LIN {X 0,Y 130.565,Z 392.696,A -85,B 0,C 180,E1 -26244.314,E2 -26244.314} C_VEL
LIN {X 0,Y 127.932,Z 388.905,A -85,B 0,C 180,E1 -26247.47,E2 -26247.47} C_VEL
LIN {X 0,Y 124.893,Z 385.428,A -85,B 0,C 180,E1 -26251.722,E2 -26251.722} C_VEL
LIN {X 0,Y 123.933,Z 383.506,A -85,B 0,C 180,E1 -26253.474,E2 -26253.474} C_VEL
LIN {X 0,Y 121.317,Z 381.44,A -85,B 0,C 180,E1 -26258.762,E2 -26258.762} C_VEL
LIN {X 0,Y 119.958,Z 378.25,A -85,B 0,C 180,E1 -26264.062,E2 -26264.062} C_VEL
LIN {X 0,Y 119.864,Z 377.879,A -85,B 0,C 180,E1 -26264.703,E2 -26264.703} C_VEL
LIN {X 0,Y 119.859,Z 377.69,A -85,B 0,C 180,E1 -26276.64,E2 -26276.64} C_VEL
LIN {X 0,Y 120.448,Z 377.843,A -85,B 0,C 180,E1 -26279.061,E2 -26279.061} C_VEL
LIN {X 0,Y 121.379,Z 380.802,A -85,B 0,C 180,E1 -26282.646,E2 -26282.646} C_VEL
LIN {X 0,Y 123.476,Z 382.974,A -85,B 0,C 180,E1 -26287.153,E2 -26287.153} C_VEL
LIN {X 0,Y 124.269,Z 383.517,A -85,B 0,C 180,E1 -26288.487,E2 -26288.487} C_VEL
LIN {X 0,Y 126.216,Z 386.94,A -85,B 0,C 180,E1 -26291.712,E2 -26291.712} C_VEL
LIN {X 0,Y 128.213,Z 389.093,A -85,B 0,C 180,E1 -26294.339,E2 -26294.339} C_VEL
LIN {X 0,Y 131.436,Z 393.757,A -85,B 0,C 180,E1 -26298.071,E2 -26298.071} C_VEL
LIN {X 0,Y 134.937,Z 398.949,A -85,B 0,C 180,E1 -26301.484,E2 -26301.484} C_VEL
LIN {X 0,Y 138.77,Z 404.783,A -85,B 0,C 180,E1 -26304.698,E2 -26304.698} C_VEL
LIN {X 0,Y 143.672,Z 413.223,A -85,B 0,C 180,E1 -26308.311,E2 -26308.311} C_VEL
LIN {X 0,Y 147.61,Z 423.228,A -85,B 0,C 180,E1 -26311.147,E2 -26311.147} C_VEL
LIN {X 0,Y 151.744,Z 435.74,A -85,B 0,C 180,E1 -26313.948,E2 -26313.948} C_VEL
LIN {X 0,Y 152.367,Z 437.977,A -85,B 0,C 180,E1 -26314.368,E2 -26314.368} C_VEL
LIN {X 0,Y 147.684,Z 494.344,A -85,B 0,C 180,E1 -26316.574,E2 -26316.574} C_VEL
LIN {X 0,Y 145.389,Z 508.708,A -85,B 0,C 180,E1 -26317.524,E2 -26317.524} C_VEL
LIN {X 0,Y 142.287,Z 522.638,A -85,B 0,C 180,E1 -26318.924,E2 -26318.924} C_VEL
LIN {X 0,Y 138.683,Z 534.674,A -85,B 0,C 180,E1 -26320.519,E2 -26320.519} C_VEL
LIN {X 0,Y 134.203,Z 547.477,A -85,B 0,C 180,E1 -26322.845,E2 -26322.845} C_VEL
LIN {X 0,Y 130.787,Z 556.168,A -85,B 0,C 180,E1 -26324.873,E2 -26324.873} C_VEL
LIN {X 0,Y 126.494,Z 565.822,A -85,B 0,C 180,E1 -26327.646,E2 -26327.646} C_VEL
LIN {X 0,Y 121.378,Z 576.257,A -85,B 0,C 180,E1 -26331.502,E2 -26331.502} C_VEL
LIN {X 0,Y 116.597,Z 585.681,A -85,B 0,C 180,E1 -26336.11,E2 -26336.11} C_VEL
LIN {X 0,Y 112.251,Z 594.067,A -85,B 0,C 180,E1 -26341.476,E2 -26341.476} C_VEL
LIN {X 0,Y 109.035,Z 600.953,A -85,B 0,C 180,E1 -26347.245,E2 -26347.245} C_VEL
LIN {X 0,Y 106.871,Z 606.138,A -85,B 0,C 180,E1 -26352.783,E2 -26352.783} C_VEL
LIN {X 0,Y 105.467,Z 611.465,A -85,B 0,C 180,E1 -26360.407,E2 -26360.407} C_VEL
LIN {X 0,Y 105.191,Z 614.408,A -85,B 0,C 180,E1 -26366.166,E2 -26366.166} C_VEL
LIN {X 0,Y 105.389,Z 615.906,A -85,B 0,C 180,E1 -26369.997,E2 -26369.997} C_VEL
LIN {X 0,Y 105.237,Z 617.007,A -85,B 0,C 180,E1 -26373.826,E2 -26373.826} C_VEL
LIN {X 0,Y 105.699,Z 618.187,A -85,B 0,C 180,E1 -26381.502,E2 -26381.502} C_VEL
LIN {X 0,Y 107.664,Z 618.07,A -85,B 0,C 180,E1 -26389.046,E2 -26389.046} C_VEL
LIN {X 0,Y 111.464,Z 616.681,A -85,B 0,C 180,E1 -26396.187,E2 -26396.187} C_VEL
LIN {X 0,Y 116.761,Z 613.987,A -85,B 0,C 180,E1 -26402.797,E2 -26402.797} C_VEL
LIN {X 0,Y 123.623,Z 609.914,A -85,B 0,C 180,E1 -26408.704,E2 -26408.704} C_VEL
LIN {X 0,Y 131.691,Z 604.349,A -85,B 0,C 180,E1 -26413.925,E2 -26413.925} C_VEL
LIN {X 0,Y 135.186,Z 601.698,A -85,B 0,C 180,E1 -26415.806,E2 -26415.806} C_VEL
LIN {X 0,Y 138.09,Z 599.07,A -85,B 0,C 180,E1 -26417.662,E2 -26417.662} C_VEL
LIN {X 0,Y 141.798,Z 594.527,A -85,B 0,C 180,E1 -26420.954,E2 -26420.954} C_VEL
LIN {X 0,Y 145.772,Z 589.525,A -85,B 0,C 180,E1 -26423.968,E2 -26423.968} C_VEL
LIN {X 0,Y 148.969,Z 586.107,A -85,B 0,C 180,E1 -26425.363,E2 -26425.363} C_VEL
LIN {X 0,Y 157.532,Z 576.958,A -85,B 0,C 180,E1 -26427.952,E2 -26427.952} C_VEL
LIN {X 0,Y 166.118,Z 566.304,A -85,B 0,C 180,E1 -26430.141,E2 -26430.141} C_VEL
LIN {X 0,Y 174.249,Z 554.394,A -85,B 0,C 180,E1 -26431.914,E2 -26431.914} C_VEL
LIN {X 0,Y 181.076,Z 542.412,A -85,B 0,C 180,E1 -26433.207,E2 -26433.207} C_VEL
LIN {X 0,Y 187.168,Z 529.101,A -85,B 0,C 180,E1 -26434.308,E2 -26434.308} C_VEL
LIN {X 0,Y 192.216,Z 515.011,A -85,B 0,C 180,E1 -26435.118,E2 -26435.118} C_VEL
LIN {X 0,Y 196.051,Z 500.312,A -85,B 0,C 180,E1 -26435.708,E2 -26435.708} C_VEL
LIN {X 0,Y 198.473,Z 485.503,A -85,B 0,C 180,E1 -26436.14,E2 -26436.14} C_VEL
LIN {X 0,Y 199.396,Z 476.925,A -85,B 0,C 180,E1 -26436.363,E2 -26436.363} C_VEL
LIN {X 0,Y 198.019,Z 472.232,A -85,B 0,C 180,E1 -26438.547,E2 -26438.547} C_VEL
LIN {X 0,Y 196.974,Z 468.88,A -85,B 0,C 180,E1 -26440.498,E2 -26440.498} C_VEL
LIN {X 0,Y 195.91,Z 465.386,A -85,B 0,C 180,E1 -26443.053,E2 -26443.053} C_VEL
LIN {X 0,Y 195.243,Z 463.284,A -85,B 0,C 180,E1 -26445.138,E2 -26445.138} C_VEL
LIN {X 0,Y 194.3,Z 461.074,A -85,B 0,C 180,E1 -26451.68,E2 -26451.68} C_VEL
LIN {X 0,Y 195.325,Z 463.03,A -85,B 0,C 180,E1 -26457.55,E2 -26457.55} C_VEL
LIN {X 0,Y 196.809,Z 466.839,A -85,B 0,C 180,E1 -26461.401,E2 -26461.401} C_VEL
LIN {X 0,Y 198.529,Z 470.876,A -85,B 0,C 180,E1 -26464.413,E2 -26464.413} C_VEL
LIN {X 0,Y 199.707,Z 473.742,A -85,B 0,C 180,E1 -26466.094,E2 -26466.094} C_VEL
LIN {X 0,Y 197.371,Z 491.479,A -85,B 0,C 180,E1 -26466.567,E2 -26466.567} C_VEL
LIN {X 0,Y 194.393,Z 504.956,A -85,B 0,C 180,E1 -26467.115,E2 -26467.115} C_VEL
LIN {X 0,Y 189.943,Z 519.303,A -85,B 0,C 180,E1 -26467.963,E2 -26467.963} C_VEL
LIN {X 0,Y 184.163,Z 533.238,A -85,B 0,C 180,E1 -26469.107,E2 -26469.107} C_VEL
LIN {X 0,Y 177.795,Z 545.567,A -85,B 0,C 180,E1 -26470.508,E2 -26470.508} C_VEL
LIN {X 0,Y 170.279,Z 557.457,A -85,B 0,C 180,E1 -26472.235,E2 -26472.235} C_VEL
LIN {X 0,Y 163.039,Z 567.153,A -85,B 0,C 180,E1 -26474.107,E2 -26474.107} C_VEL
LIN {X 0,Y 155.175,Z 576.173,A -85,B 0,C 180,E1 -26476.356,E2 -26476.356} C_VEL
LIN {X 0,Y 146.298,Z 584.96,A -85,B 0,C 180,E1 -26479.346,E2 -26479.346} C_VEL
LIN {X 0,Y 137.329,Z 592.535,A -85,B 0,C 180,E1 -26482.91,E2 -26482.91} C_VEL
LIN {X 0,Y 129.687,Z 598.111,A -85,B 0,C 180,E1 -26486.606,E2 -26486.606} C_VEL
LIN {X 0,Y 121.78,Z 603.078,A -85,B 0,C 180,E1 -26491.29,E2 -26491.29} C_VEL
LIN {X 0,Y 114.351,Z 606.986,A -85,B 0,C 180,E1 -26496.973,E2 -26496.973} C_VEL
LIN {X 0,Y 107.549,Z 609.772,A -85,B 0,C 180,E1 -26504.048,E2 -26504.048} C_VEL
LIN {X 0,Y 102.478,Z 611.008,A -85,B 0,C 180,E1 -26511.891,E2 -26511.891} C_VEL
LIN {X 0,Y 99.227,Z 610.742,A -85,B 0,C 180,E1 -26520.282,E2 -26520.282} C_VEL
LIN {X 0,Y 97.751,Z 608.962,A -85,B 0,C 180,E1 -26529.17,E2 -26529.17} C_VEL
LIN {X 0,Y 97.864,Z 605.87,A -85,B 0,C 180,E1 -26537.562,E2 -26537.562} C_VEL
LIN {X 0,Y 98.97,Z 602.563,A -85,B 0,C 180,E1 -26543.788,E2 -26543.788} C_VEL
LIN {X 0,Y 100.796,Z 598.268,A -85,B 0,C 180,E1 -26550.004,E2 -26550.004} C_VEL
LIN {X 0,Y 103.829,Z 592.06,A -85,B 0,C 180,E1 -26556.806,E2 -26556.806} C_VEL
LIN {X 0,Y 107.94,Z 584.679,A -85,B 0,C 180,E1 -26562.874,E2 -26562.874} C_VEL
LIN {X 0,Y 112.553,Z 576.205,A -85,B 0,C 180,E1 -26568.196,E2 -26568.196} C_VEL
LIN {X 0,Y 117.725,Z 566.442,A -85,B 0,C 180,E1 -26572.836,E2 -26572.836} C_VEL
LIN {X 0,Y 123.092,Z 555.588,A -85,B 0,C 180,E1 -26576.723,E2 -26576.723} C_VEL
LIN {X 0,Y 128.33,Z 543.576,A -85,B 0,C 180,E1 -26579.985,E2 -26579.985} C_VEL
LIN {X 0,Y 133.128,Z 530.85,A -85,B 0,C 180,E1 -26582.567,E2 -26582.567} C_VEL
LIN {X 0,Y 137.139,Z 517.829,A -85,B 0,C 180,E1 -26584.539,E2 -26584.539} C_VEL
LIN {X 0,Y 140.486,Z 503.558,A -85,B 0,C 180,E1 -26586.115,E2 -26586.115} C_VEL
LIN {X 0,Y 142.816,Z 489.892,A -85,B 0,C 180,E1 -26587.138,E2 -26587.138} C_VEL
LIN {X 0,Y 144.553,Z 473.342,A -85,B 0,C 180,E1 -26587.883,E2 -26587.883} C_VEL
LIN {X 0,Y 147.842,Z 434.546,A -85,B 0,C 180,E1 -26589.335,E2 -26589.335} C_VEL
LIN {X 0,Y 143.5,Z 424.674,A -85,B 0,C 180,E1 -26592.28,E2 -26592.28} C_VEL
LIN {X 0,Y 138.696,Z 415.374,A -85,B 0,C 180,E1 -26595.804,E2 -26595.804} C_VEL
LIN {X 0,Y 133.828,Z 407.051,A -85,B 0,C 180,E1 -26599.922,E2 -26599.922} C_VEL
LIN {X 0,Y 130.389,Z 401.996,A -85,B 0,C 180,E1 -26603.29,E2 -26603.29} C_VEL
LIN {X 0,Y 128.308,Z 398.785,A -85,B 0,C 180,E1 -26605.658,E2 -26605.658} C_VEL
LIN {X 0,Y 125.687,Z 394.914,A -85,B 0,C 180,E1 -26609.089,E2 -26609.089} C_VEL
LIN {X 0,Y 123.305,Z 392.01,A -85,B 0,C 180,E1 -26612.724,E2 -26612.724} C_VEL
LIN {X 0,Y 122.54,Z 390.343,A -85,B 0,C 180,E1 -26614.234,E2 -26614.234} C_VEL
LIN {X 0,Y 120.138,Z 388.287,A -85,B 0,C 180,E1 -26619.453,E2 -26619.453} C_VEL
LIN {X 0,Y 118.826,Z 384.875,A -85,B 0,C 180,E1 -26625.443,E2 -26625.443} C_VEL
LIN {X 0,Y 119.141,Z 384.732,A -85,B 0,C 180,E1 -26637.465,E2 -26637.465} C_VEL
LIN {X 0,Y 119.373,Z 385.115,A -85,B 0,C 180,E1 -26638.563,E2 -26638.563} C_VEL
LIN {X 0,Y 120.443,Z 388.08,A -85,B 0,C 180,E1 -26642.666,E2 -26642.666} C_VEL
LIN {X 0,Y 122.798,Z 390.406,A -85,B 0,C 180,E1 -26647.639,E2 -26647.639} C_VEL
LIN {X 0,Y 124.835,Z 393.821,A -85,B 0,C 180,E1 -26651.142,E2 -26651.142} C_VEL
LIN {X 0,Y 126.414,Z 395.654,A -85,B 0,C 180,E1 -26653.346,E2 -26653.346} C_VEL
LIN {X 0,Y 129.348,Z 400.172,A -85,B 0,C 180,E1 -26657.001,E2 -26657.001} C_VEL
LIN {X 0,Y 132.297,Z 404.722,A -85,B 0,C 180,E1 -26660.1,E2 -26660.1} C_VEL
LIN {X 0,Y 135.761,Z 410.198,A -85,B 0,C 180,E1 -26663.251,E2 -26663.251} C_VEL
LIN {X 0,Y 140.215,Z 418.181,A -85,B 0,C 180,E1 -26666.816,E2 -26666.816} C_VEL
LIN {X 0,Y 143.851,Z 427.962,A -85,B 0,C 180,E1 -26669.649,E2 -26669.649} C_VEL
LIN {X 0,Y 147.514,Z 439.791,A -85,B 0,C 180,E1 -26672.38,E2 -26672.38} C_VEL
LIN {X 0,Y 142.873,Z 493.821,A -85,B 0,C 180,E1 -26674.515,E2 -26674.515} C_VEL
LIN {X 0,Y 140.487,Z 508.265,A -85,B 0,C 180,E1 -26675.46,E2 -26675.46} C_VEL
LIN {X 0,Y 137.276,Z 522.25,A -85,B 0,C 180,E1 -26676.872,E2 -26676.872} C_VEL
LIN {X 0,Y 132.944,Z 536.105,A -85,B 0,C 180,E1 -26678.759,E2 -26678.759} C_VEL
LIN {X 0,Y 128.467,Z 548.145,A -85,B 0,C 180,E1 -26681.033,E2 -26681.033} C_VEL
LIN {X 0,Y 123.348,Z 559.998,A -85,B 0,C 180,E1 -26683.996,E2 -26683.996} C_VEL
LIN {X 0,Y 117.775,Z 571.436,A -85,B 0,C 180,E1 -26687.827,E2 -26687.827} C_VEL
LIN {X 0,Y 112.305,Z 581.637,A -85,B 0,C 180,E1 -26692.396,E2 -26692.396} C_VEL
LIN {X 0,Y 107.744,Z 590.107,A -85,B 0,C 180,E1 -26697.439,E2 -26697.439} C_VEL
LIN {X 0,Y 103.985,Z 597.14,A -85,B 0,C 180,E1 -26702.854,E2 -26702.854} C_VEL
LIN {X 0,Y 100.736,Z 603.799,A -85,B 0,C 180,E1 -26709.58,E2 -26709.58} C_VEL
LIN {X 0,Y 98.674,Z 609.674,A -85,B 0,C 180,E1 -26717.659,E2 -26717.659} C_VEL
LIN {X 0,Y 98.264,Z 611.989,A -85,B 0,C 180,E1 -26721.772,E2 -26721.772} C_VEL
LIN {X 0,Y 98.308,Z 615.447,A -85,B 0,C 180,E1 -26729.996,E2 -26729.996} C_VEL
LIN {X 0,Y 98.155,Z 616.589,A -85,B 0,C 180,E1 -26734.102,E2 -26734.102} C_VEL
LIN {X 0,Y 98.71,Z 617.854,A -85,B 0,C 180,E1 -26742.329,E2 -26742.329} C_VEL
LIN {X 0,Y 100.934,Z 617.823,A -85,B 0,C 180,E1 -26750.37,E2 -26750.37} C_VEL
LIN {X 0,Y 105.094,Z 616.524,A -85,B 0,C 180,E1 -26757.908,E2 -26757.908} C_VEL
LIN {X 0,Y 110.842,Z 613.932,A -85,B 0,C 180,E1 -26764.791,E2 -26764.791} C_VEL
LIN {X 0,Y 118.143,Z 609.985,A -85,B 0,C 180,E1 -26770.867,E2 -26770.867} C_VEL
LIN {X 0,Y 126.657,Z 604.538,A -85,B 0,C 180,E1 -26776.161,E2 -26776.161} C_VEL
LIN {X 0,Y 133.774,Z 599.397,A -85,B 0,C 180,E1 -26779.616,E2 -26779.616} C_VEL
LIN {X 0,Y 142.665,Z 592.072,A -85,B 0,C 180,E1 -26783.174,E2 -26783.174} C_VEL
LIN {X 0,Y 148.969,Z 586.107,A -85,B 0,C 180,E1 -26785.363,E2 -26785.363} C_VEL
LIN {X 0,Y 152.163,Z 582.553,A -85,B 0,C 180,E1 -26786.685,E2 -26786.685} C_VEL
LIN {X 0,Y 156.304,Z 576.602,A -85,B 0,C 180,E1 -26789.221,E2 -26789.221} C_VEL
LIN {X 0,Y 160.479,Z 570.287,A -85,B 0,C 180,E1 -26791.519,E2 -26791.519} C_VEL
LIN {X 0,Y 163.59,Z 566.039,A -85,B 0,C 180,E1 -26792.464,E2 -26792.464} C_VEL
LIN {X 0,Y 171.828,Z 554.28,A -85,B 0,C 180,E1 -26794.13,E2 -26794.13} C_VEL
LIN {X 0,Y 178.803,Z 542.339,A -85,B 0,C 180,E1 -26795.354,E2 -26795.354} C_VEL
LIN {X 0,Y 185.017,Z 529.103,A -85,B 0,C 180,E1 -26796.4,E2 -26796.4} C_VEL
LIN {X 0,Y 190.172,Z 515.088,A -85,B 0,C 180,E1 -26797.154,E2 -26797.154} C_VEL
LIN {X 0,Y 193.988,Z 500.922,A -85,B 0,C 180,E1 -26797.696,E2 -26797.696} C_VEL
LIN {X 0,Y 196.522,Z 486.259,A -85,B 0,C 180,E1 -26798.109,E2 -26798.109} C_VEL
LIN {X 0,Y 197.129,Z 480.708,A -85,B 0,C 180,E1 -26798.293,E2 -26798.293} C_VEL
LIN {X 0,Y 195.702,Z 475.495,A -85,B 0,C 180,E1 -26801.142,E2 -26801.142} C_VEL
LIN {X 0,Y 194.724,Z 471.967,A -85,B 0,C 180,E1 -26803.756,E2 -26803.756} C_VEL
LIN {X 0,Y 194.117,Z 470.099,A -85,B 0,C 180,E1 -26805.854,E2 -26805.854} C_VEL
LIN {X 0,Y 193.405,Z 468.125,A -85,B 0,C 180,E1 -26811.642,E2 -26811.642} C_VEL
LIN {X 0,Y 194.291,Z 469.945,A -85,B 0,C 180,E1 -26817.148,E2 -26817.148} C_VEL
LIN {X 0,Y 195.675,Z 473.82,A -85,B 0,C 180,E1 -26821.02,E2 -26821.02} C_VEL
LIN {X 0,Y 197.375,Z 478.057,A -85,B 0,C 180,E1 -26824.16,E2 -26824.16} C_VEL
LIN {X 0,Y 195.492,Z 491.681,A -85,B 0,C 180,E1 -26824.575,E2 -26824.575} C_VEL
LIN {X 0,Y 192.282,Z 505.823,A -85,B 0,C 180,E1 -26825.124,E2 -26825.124} C_VEL
LIN {X 0,Y 187.68,Z 520.146,A -85,B 0,C 180,E1 -26825.946,E2 -26825.946} C_VEL
LIN {X 0,Y 182.297,Z 532.862,A -85,B 0,C 180,E1 -26826.935,E2 -26826.935} C_VEL
LIN {X 0,Y 175.759,Z 545.305,A -85,B 0,C 180,E1 -26828.262,E2 -26828.262} C_VEL
LIN {X 0,Y 168.052,Z 557.274,A -85,B 0,C 180,E1 -26829.909,E2 -26829.909} C_VEL
LIN {X 0,Y 159.79,Z 567.991,A -85,B 0,C 180,E1 -26831.884,E2 -26831.884} C_VEL
LIN {X 0,Y 152.067,Z 576.524,A -85,B 0,C 180,E1 -26833.953,E2 -26833.953} C_VEL
LIN {X 0,Y 143.374,Z 584.837,A -85,B 0,C 180,E1 -26836.675,E2 -26836.675} C_VEL
LIN {X 0,Y 134.546,Z 592.07,A -85,B 0,C 180,E1 -26839.92,E2 -26839.92} C_VEL
LIN {X 0,Y 126.152,Z 597.976,A -85,B 0,C 180,E1 -26843.63,E2 -26843.63} C_VEL
LIN {X 0,Y 116.987,Z 603.443,A -85,B 0,C 180,E1 -26848.723,E2 -26848.723} C_VEL
LIN {X 0,Y 109.905,Z 606.939,A -85,B 0,C 180,E1 -26853.774,E2 -26853.774} C_VEL
LIN {X 0,Y 102.361,Z 609.85,A -85,B 0,C 180,E1 -26860.959,E2 -26860.959} C_VEL
LIN {X 0,Y 96.569,Z 611.237,A -85,B 0,C 180,E1 -26869.086,E2 -26869.086} C_VEL
LIN {X 0,Y 92.708,Z 611.122,A -85,B 0,C 180,E1 -26877.955,E2 -26877.955} C_VEL
LIN {X 0,Y 90.794,Z 609.529,A -85,B 0,C 180,E1 -26887.235,E2 -26887.235} C_VEL
LIN {X 0,Y 90.662,Z 606.49,A -85,B 0,C 180,E1 -26896.557,E2 -26896.557} C_VEL
LIN {X 0,Y 91.859,Z 602.883,A -85,B 0,C 180,E1 -26904.033,E2 -26904.033} C_VEL
LIN {X 0,Y 94.334,Z 597.49,A -85,B 0,C 180,E1 -26912.139,E2 -26912.139} C_VEL
LIN {X 0,Y 97.853,Z 591.02,A -85,B 0,C 180,E1 -26919.303,E2 -26919.303} C_VEL
LIN {X 0,Y 102.587,Z 582.975,A -85,B 0,C 180,E1 -26925.908,E2 -26925.908} C_VEL
LIN {X 0,Y 107.51,Z 574.56,A -85,B 0,C 180,E1 -26931.075,E2 -26931.075} C_VEL
LIN {X 0,Y 113.086,Z 564.432,A -85,B 0,C 180,E1 -26935.791,E2 -26935.791} C_VEL
LIN {X 0,Y 118.876,Z 553.081,A -85,B 0,C 180,E1 -26939.682,E2 -26939.682} C_VEL
LIN {X 0,Y 123.921,Z 541.774,A -85,B 0,C 180,E1 -26942.604,E2 -26942.604} C_VEL
LIN {X 0,Y 128.938,Z 528.539,A -85,B 0,C 180,E1 -26945.156,E2 -26945.156} C_VEL
LIN {X 0,Y 133.138,Z 514.65,A -85,B 0,C 180,E1 -26947.143,E2 -26947.143} C_VEL
LIN {X 0,Y 136.364,Z 500.569,A -85,B 0,C 180,E1 -26948.583,E2 -26948.583} C_VEL
LIN {X 0,Y 138.668,Z 486.383,A -85,B 0,C 180,E1 -26949.526,E2 -26949.526} C_VEL
LIN {X 0,Y 143.173,Z 436.992,A -85,B 0,C 180,E1 -26951.425,E2 -26951.425} C_VEL
LIN {X 0,Y 138.636,Z 426.756,A -85,B 0,C 180,E1 -26954.79,E2 -26954.79} C_VEL
LIN {X 0,Y 134.385,Z 418.447,A -85,B 0,C 180,E1 -26958.313,E2 -26958.313} C_VEL
LIN {X 0,Y 130.256,Z 411.423,A -85,B 0,C 180,E1 -26962.248,E2 -26962.248} C_VEL
LIN {X 0,Y 126.452,Z 405.272,A -85,B 0,C 180,E1 -26966.64,E2 -26966.64} C_VEL
LIN {X 0,Y 123.842,Z 401.369,A -85,B 0,C 180,E1 -26970.293,E2 -26970.293} C_VEL
LIN {X 0,Y 121.463,Z 398.016,A -85,B 0,C 180,E1 -26974.334,E2 -26974.334} C_VEL
LIN {X 0,Y 121.025,Z 397.131,A -85,B 0,C 180,E1 -26975.272,E2 -26975.272} C_VEL
LIN {X 0,Y 118.602,Z 394.472,A -85,B 0,C 180,E1 -26981.47,E2 -26981.47} C_VEL
LIN {X 0,Y 117.811,Z 391.858,A -85,B 0,C 180,E1 -26986.196,E2 -26986.196} C_VEL
LIN {X 0,Y 118.259,Z 391.878,A -85,B 0,C 180,E1 -26997.603,E2 -26997.603} C_VEL
LIN {X 0,Y 119.232,Z 394.875,A -85,B 0,C 180,E1 -27001.872,E2 -27001.872} C_VEL
LIN {X 0,Y 121.348,Z 397.207,A -85,B 0,C 180,E1 -27006.751,E2 -27006.751} C_VEL
LIN {X 0,Y 123.458,Z 400.701,A -85,B 0,C 180,E1 -27010.55,E2 -27010.55} C_VEL
LIN {X 0,Y 124.654,Z 402.238,A -85,B 0,C 180,E1 -27012.33,E2 -27012.33} C_VEL
LIN {X 0,Y 127.406,Z 406.711,A -85,B 0,C 180,E1 -27016.011,E2 -27016.011} C_VEL
LIN {X 0,Y 130.249,Z 411.318,A -85,B 0,C 180,E1 -27019.198,E2 -27019.198} C_VEL
LIN {X 0,Y 133.511,Z 416.904,A -85,B 0,C 180,E1 -27022.367,E2 -27022.367} C_VEL
LIN {X 0,Y 136.961,Z 423.54,A -85,B 0,C 180,E1 -27025.351,E2 -27025.351} C_VEL
LIN {X 0,Y 140.042,Z 432.268,A -85,B 0,C 180,E1 -27027.965,E2 -27027.965} C_VEL
LIN {X 0,Y 142.868,Z 441.747,A -85,B 0,C 180,E1 -27030.281,E2 -27030.281} C_VEL
LIN {X 0,Y 138.312,Z 492.874,A -85,B 0,C 180,E1 -27032.288,E2 -27032.288} C_VEL
LIN {X 0,Y 135.883,Z 507.41,A -85,B 0,C 180,E1 -27033.223,E2 -27033.223} C_VEL
LIN {X 0,Y 132.455,Z 521.863,A -85,B 0,C 180,E1 -27034.668,E2 -27034.668} C_VEL
LIN {X 0,Y 127.952,Z 535.743,A -85,B 0,C 180,E1 -27036.549,E2 -27036.549} C_VEL
LIN {X 0,Y 123.17,Z 548.031,A -85,B 0,C 180,E1 -27038.878,E2 -27038.878} C_VEL
LIN {X 0,Y 117.914,Z 559.668,A -85,B 0,C 180,E1 -27041.834,E2 -27041.834} C_VEL
LIN {X 0,Y 112.578,Z 570.177,A -85,B 0,C 180,E1 -27045.383,E2 -27045.383} C_VEL
LIN {X 0,Y 106.709,Z 580.573,A -85,B 0,C 180,E1 -27050.044,E2 -27050.044} C_VEL
LIN {X 0,Y 101.75,Z 589.176,A -85,B 0,C 180,E1 -27055.257,E2 -27055.257} C_VEL
LIN {X 0,Y 97.059,Z 597.36,A -85,B 0,C 180,E1 -27061.919,E2 -27061.919} C_VEL
LIN {X 0,Y 94.071,Z 603.1,A -85,B 0,C 180,E1 -27068.061,E2 -27068.061} C_VEL
LIN {X 0,Y 91.718,Z 609.076,A -85,B 0,C 180,E1 -27076.706,E2 -27076.706} C_VEL
LIN {X 0,Y 91.217,Z 611.437,A -85,B 0,C 180,E1 -27081.132,E2 -27081.132} C_VEL
LIN {X 0,Y 91.217,Z 614.987,A -85,B 0,C 180,E1 -27089.996,E2 -27089.996} C_VEL
LIN {X 0,Y 91.066,Z 616.171,A -85,B 0,C 180,E1 -27094.422,E2 -27094.422} C_VEL
LIN {X 0,Y 91.757,Z 617.52,A -85,B 0,C 180,E1 -27103.28,E2 -27103.28} C_VEL
LIN {X 0,Y 94.267,Z 617.573,A -85,B 0,C 180,E1 -27111.882,E2 -27111.882} C_VEL
LIN {X 0,Y 98.832,Z 616.364,A -85,B 0,C 180,E1 -27119.848,E2 -27119.848} C_VEL
LIN {X 0,Y 105.074,Z 613.869,A -85,B 0,C 180,E1 -27127.007,E2 -27127.007} C_VEL
LIN {X 0,Y 112.855,Z 610.028,A -85,B 0,C 180,E1 -27133.232,E2 -27133.232} C_VEL
LIN {X 0,Y 121.833,Z 604.723,A -85,B 0,C 180,E1 -27138.577,E2 -27138.577} C_VEL
LIN {X 0,Y 129.296,Z 599.641,A -85,B 0,C 180,E1 -27142.009,E2 -27142.009} C_VEL
LIN {X 0,Y 138.528,Z 592.437,A -85,B 0,C 180,E1 -27145.524,E2 -27145.524} C_VEL
LIN {X 0,Y 148.166,Z 583.599,A -85,B 0,C 180,E1 -27148.622,E2 -27148.622} C_VEL
LIN {X 0,Y 156.862,Z 574.366,A -85,B 0,C 180,E1 -27150.882,E2 -27150.882} C_VEL
LIN {X 0,Y 163.59,Z 566.039,A -85,B 0,C 180,E1 -27152.464,E2 -27152.464} C_VEL
LIN {X 0,Y 166.673,Z 561.678,A -85,B 0,C 180,E1 -27153.335,E2 -27153.335} C_VEL
LIN {X 0,Y 170.722,Z 554.474,A -85,B 0,C 180,E1 -27155.189,E2 -27155.189} C_VEL
LIN {X 0,Y 174.448,Z 546.9,A -85,B 0,C 180,E1 -27156.911,E2 -27156.911} C_VEL
LIN {X 0,Y 176.941,Z 541.962,A -85,B 0,C 180,E1 -27157.582,E2 -27157.582} C_VEL
LIN {X 0,Y 183.124,Z 529.102,A -85,B 0,C 180,E1 -27158.534,E2 -27158.534} C_VEL
LIN {X 0,Y 188.332,Z 515.305,A -85,B 0,C 180,E1 -27159.223,E2 -27159.223} C_VEL
LIN {X 0,Y 192.356,Z 500.713,A -85,B 0,C 180,E1 -27159.757,E2 -27159.757} C_VEL
LIN {X 0,Y 194.963,Z 485.994,A -85,B 0,C 180,E1 -27160.146,E2 -27160.146} C_VEL
LIN {X 0,Y 195.085,Z 484.899,A -85,B 0,C 180,E1 -27160.213,E2 -27160.213} C_VEL
LIN {X 0,Y 194.284,Z 481.515,A -85,B 0,C 180,E1 -27162.228,E2 -27162.228} C_VEL
LIN {X 0,Y 193.496,Z 478.254,A -85,B 0,C 180,E1 -27164.732,E2 -27164.732} C_VEL
LIN {X 0,Y 193.088,Z 477.008,A -85,B 0,C 180,E1 -27166.314,E2 -27166.314} C_VEL
LIN {X 0,Y 192.509,Z 475.192,A -85,B 0,C 180,E1 -27171.602,E2 -27171.602} C_VEL
LIN {X 0,Y 193.266,Z 476.862,A -85,B 0,C 180,E1 -27176.742,E2 -27176.742} C_VEL
LIN {X 0,Y 194.452,Z 480.465,A -85,B 0,C 180,E1 -27180.388,E2 -27180.388} C_VEL
LIN {X 0,Y 195.276,Z 482.796,A -85,B 0,C 180,E1 -27182.255,E2 -27182.255} C_VEL
LIN {X 0,Y 193.115,Z 495.782,A -85,B 0,C 180,E1 -27182.652,E2 -27182.652} C_VEL
LIN {X 0,Y 189.61,Z 509.454,A -85,B 0,C 180,E1 -27183.231,E2 -27183.231} C_VEL
LIN {X 0,Y 184.926,Z 522.764,A -85,B 0,C 180,E1 -27183.992,E2 -27183.992} C_VEL
LIN {X 0,Y 178.766,Z 536.319,A -85,B 0,C 180,E1 -27185.058,E2 -27185.058} C_VEL
LIN {X 0,Y 172.336,Z 547.773,A -85,B 0,C 180,E1 -27186.287,E2 -27186.287} C_VEL
LIN {X 0,Y 164.387,Z 559.452,A -85,B 0,C 180,E1 -27187.876,E2 -27187.876} C_VEL
LIN {X 0,Y 155.49,Z 570.334,A -85,B 0,C 180,E1 -27189.883,E2 -27189.883} C_VEL
LIN {X 0,Y 147.286,Z 578.835,A -85,B 0,C 180,E1 -27192.002,E2 -27192.002} C_VEL
LIN {X 0,Y 138.081,Z 587.013,A -85,B 0,C 180,E1 -27194.759,E2 -27194.759} C_VEL
LIN {X 0,Y 129.239,Z 593.716,A -85,B 0,C 180,E1 -27197.901,E2 -27197.901} C_VEL
LIN {X 0,Y 120.837,Z 599.162,A -85,B 0,C 180,E1 -27201.485,E2 -27201.485} C_VEL
LIN {X 0,Y 112.414,Z 603.82,A -85,B 0,C 180,E1 -27205.952,E2 -27205.952} C_VEL
LIN {X 0,Y 105.827,Z 606.892,A -85,B 0,C 180,E1 -27210.314,E2 -27210.314} C_VEL
LIN {X 0,Y 97.49,Z 609.929,A -85,B 0,C 180,E1 -27217.541,E2 -27217.541} C_VEL
LIN {X 0,Y 90.922,Z 611.436,A -85,B 0,C 180,E1 -27225.925,E2 -27225.925} C_VEL
LIN {X 0,Y 86.377,Z 611.466,A -85,B 0,C 180,E1 -27235.287,E2 -27235.287} C_VEL
LIN {X 0,Y 83.897,Z 610.021,A -85,B 0,C 180,E1 -27245.243,E2 -27245.243} C_VEL
LIN {X 0,Y 83.44,Z 608.743,A -85,B 0,C 180,E1 -27250.316,E2 -27250.316} C_VEL
LIN {X 0,Y 84.053,Z 605.08,A -85,B 0,C 180,E1 -27260.378,E2 -27260.378} C_VEL
LIN {X 0,Y 85.594,Z 601.369,A -85,B 0,C 180,E1 -27267.651,E2 -27267.651} C_VEL
LIN {X 0,Y 87.992,Z 596.701,A -85,B 0,C 180,E1 -27274.585,E2 -27274.585} C_VEL
LIN {X 0,Y 92.051,Z 589.969,A -85,B 0,C 180,E1 -27282.124,E2 -27282.124} C_VEL
LIN {X 0,Y 97.368,Z 581.584,A -85,B 0,C 180,E1 -27288.958,E2 -27288.958} C_VEL
LIN {X 0,Y 102.738,Z 572.829,A -85,B 0,C 180,E1 -27294.236,E2 -27294.236} C_VEL
LIN {X 0,Y 108.804,Z 562.214,A -85,B 0,C 180,E1 -27298.98,E2 -27298.98} C_VEL
LIN {X 0,Y 114.423,Z 551.482,A -85,B 0,C 180,E1 -27302.513,E2 -27302.513} C_VEL
LIN {X 0,Y 119.788,Z 539.763,A -85,B 0,C 180,E1 -27305.41,E2 -27305.41} C_VEL
LIN {X 0,Y 124.798,Z 526.675,A -85,B 0,C 180,E1 -27307.834,E2 -27307.834} C_VEL
LIN {X 0,Y 128.809,Z 513.594,A -85,B 0,C 180,E1 -27309.623,E2 -27309.623} C_VEL
LIN {X 0,Y 132.1,Z 499.36,A -85,B 0,C 180,E1 -27311.023,E2 -27311.023} C_VEL
LIN {X 0,Y 134.414,Z 484.873,A -85,B 0,C 180,E1 -27311.907,E2 -27311.907} C_VEL
LIN {X 0,Y 138.632,Z 439.572,A -85,B 0,C 180,E1 -27313.64,E2 -27313.64} C_VEL
LIN {X 0,Y 134.588,Z 430.258,A -85,B 0,C 180,E1 -27316.979,E2 -27316.979} C_VEL
LIN {X 0,Y 131.132,Z 423.275,A -85,B 0,C 180,E1 -27320.17,E2 -27320.17} C_VEL
LIN {X 0,Y 127.804,Z 417.282,A -85,B 0,C 180,E1 -27323.668,E2 -27323.668} C_VEL
LIN {X 0,Y 124.306,Z 411.372,A -85,B 0,C 180,E1 -27328.086,E2 -27328.086} C_VEL
LIN {X 0,Y 122.054,Z 407.807,A -85,B 0,C 180,E1 -27331.503,E2 -27331.503} C_VEL
LIN {X 0,Y 119.818,Z 404.229,A -85,B 0,C 180,E1 -27335.76,E2 -27335.76} C_VEL
LIN {X 0,Y 117.128,Z 400.289,A -85,B 0,C 180,E1 -27344.113,E2 -27344.113} C_VEL
LIN {X 0,Y 116.912,Z 399.034,A -85,B 0,C 180,E1 -27346.088,E2 -27346.088} C_VEL
LIN {X 0,Y 116.679,Z 398.767,A -85,B 0,C 180,E1 -27353.082,E2 -27353.082} C_VEL
LIN {X 0,Y 117.23,Z 398.988,A -85,B 0,C 180,E1 -27357.076,E2 -27357.076} C_VEL
LIN {X 0,Y 118.365,Z 402.176,A -85,B 0,C 180,E1 -27362.07,E2 -27362.07} C_VEL
LIN {X 0,Y 119.958,Z 404.022,A -85,B 0,C 180,E1 -27365.896,E2 -27365.896} C_VEL
LIN {X 0,Y 122.086,Z 407.575,A -85,B 0,C 180,E1 -27369.946,E2 -27369.946} C_VEL
LIN {X 0,Y 123.233,Z 409.368,A -85,B 0,C 180,E1 -27371.762,E2 -27371.762} C_VEL
LIN {X 0,Y 125.272,Z 412.815,A -85,B 0,C 180,E1 -27374.683,E2 -27374.683} C_VEL
LIN {X 0,Y 129.08,Z 419.282,A -85,B 0,C 180,E1 -27379.172,E2 -27379.172} C_VEL
LIN {X 0,Y 133.423,Z 427.795,A -85,B 0,C 180,E1 -27383.445,E2 -27383.445} C_VEL
LIN {X 0,Y 136.155,Z 435.921,A -85,B 0,C 180,E1 -27386.025,E2 -27386.025} C_VEL
LIN {X 0,Y 138.391,Z 443.732,A -85,B 0,C 180,E1 -27388.049,E2 -27388.049} C_VEL
LIN {X 0,Y 133.809,Z 492.939,A -85,B 0,C 180,E1 -27389.976,E2 -27389.976} C_VEL
LIN {X 0,Y 131.395,Z 506.941,A -85,B 0,C 180,E1 -27390.869,E2 -27390.869} C_VEL
LIN {X 0,Y 128.178,Z 520.287,A -85,B 0,C 180,E1 -27392.169,E2 -27392.169} C_VEL
LIN {X 0,Y 123.794,Z 533.546,A -85,B 0,C 180,E1 -27393.867,E2 -27393.867} C_VEL
LIN {X 0,Y 118.56,Z 546.785,A -85,B 0,C 180,E1 -27396.307,E2 -27396.307} C_VEL
LIN {X 0,Y 114.463,Z 555.749,A -85,B 0,C 180,E1 -27398.474,E2 -27398.474} C_VEL
LIN {X 0,Y 109.242,Z 565.875,A -85,B 0,C 180,E1 -27401.588,E2 -27401.588} C_VEL
LIN {X 0,Y 103.293,Z 576.149,A -85,B 0,C 180,E1 -27405.777,E2 -27405.777} C_VEL
LIN {X 0,Y 97.623,Z 585.459,A -85,B 0,C 180,E1 -27410.951,E2 -27410.951} C_VEL
LIN {X 0,Y 92.634,Z 593.359,A -85,B 0,C 180,E1 -27416.833,E2 -27416.833} C_VEL
LIN {X 0,Y 88.455,Z 600.536,A -85,B 0,C 180,E1 -27424.084,E2 -27424.084} C_VEL
LIN {X 0,Y 85.834,Z 605.65,A -85,B 0,C 180,E1 -27430.878,E2 -27430.878} C_VEL
LIN {X 0,Y 84.422,Z 609.734,A -85,B 0,C 180,E1 -27437.983,E2 -27437.983} C_VEL
LIN {X 0,Y 83.918,Z 612.893,A -85,B 0,C 180,E1 -27445.192,E2 -27445.192} C_VEL
LIN {X 0,Y 84.133,Z 614.527,A -85,B 0,C 180,E1 -27449.996,E2 -27449.996} C_VEL
LIN {X 0,Y 83.979,Z 615.752,A -85,B 0,C 180,E1 -27454.796,E2 -27454.796} C_VEL
LIN {X 0,Y 84.845,Z 617.183,A -85,B 0,C 180,E1 -27464.384,E2 -27464.384} C_VEL
LIN {X 0,Y 87.683,Z 617.326,A -85,B 0,C 180,E1 -27473.621,E2 -27473.621} C_VEL
LIN {X 0,Y 92.702,Z 616.207,A -85,B 0,C 180,E1 -27482.047,E2 -27482.047} C_VEL
LIN {X 0,Y 99.465,Z 613.805,A -85,B 0,C 180,E1 -27489.483,E2 -27489.483} C_VEL
LIN {X 0,Y 107.763,Z 610.061,A -85,B 0,C 180,E1 -27495.834,E2 -27495.834} C_VEL
LIN {X 0,Y 117.244,Z 604.869,A -85,B 0,C 180,E1 -27501.187,E2 -27501.187} C_VEL
LIN {X 0,Y 125.051,Z 599.885,A -85,B 0,C 180,E1 -27504.573,E2 -27504.573} C_VEL
LIN {X 0,Y 134.64,Z 592.801,A -85,B 0,C 180,E1 -27508.013,E2 -27508.013} C_VEL
LIN {X 0,Y 144.609,Z 584.098,A -85,B 0,C 180,E1 -27511.016,E2 -27511.016} C_VEL
LIN {X 0,Y 153.553,Z 575.021,A -85,B 0,C 180,E1 -27513.183,E2 -27513.183} C_VEL
LIN {X 0,Y 161.135,Z 566.025,A -85,B 0,C 180,E1 -27514.82,E2 -27514.82} C_VEL
LIN {X 0,Y 168.871,Z 555.335,A -85,B 0,C 180,E1 -27516.283,E2 -27516.283} C_VEL
LIN {X 0,Y 175.993,Z 543.672,A -85,B 0,C 180,E1 -27517.431,E2 -27517.431} C_VEL
LIN {X 0,Y 176.941,Z 541.962,A -85,B 0,C 180,E1 -27517.582,E2 -27517.582} C_VEL
LIN {X 0,Y 179.343,Z 536.914,A -85,B 0,C 180,E1 -27518.208,E2 -27518.208} C_VEL
LIN {X 0,Y 182.52,Z 528.676,A -85,B 0,C 180,E1 -27519.643,E2 -27519.643} C_VEL
LIN {X 0,Y 185.325,Z 520.178,A -85,B 0,C 180,E1 -27520.943,E2 -27520.943} C_VEL
LIN {X 0,Y 187.066,Z 514.732,A -85,B 0,C 180,E1 -27521.369,E2 -27521.369} C_VEL
LIN {X 0,Y 191.015,Z 500.625,A -85,B 0,C 180,E1 -27521.845,E2 -27521.845} C_VEL
LIN {X 0,Y 193.208,Z 489.207,A -85,B 0,C 180,E1 -27522.168,E2 -27522.168} C_VEL
LIN {X 0,Y 192.408,Z 485.119,A -85,B 0,C 180,E1 -27525.185,E2 -27525.185} C_VEL
LIN {X 0,Y 192.063,Z 483.894,A -85,B 0,C 180,E1 -27526.779,E2 -27526.779} C_VEL
LIN {X 0,Y 191.612,Z 482.262,A -85,B 0,C 180,E1 -27531.563,E2 -27531.563} C_VEL
LIN {X 0,Y 192.214,Z 483.761,A -85,B 0,C 180,E1 -27536.331,E2 -27536.331} C_VEL
LIN {X 0,Y 193.123,Z 487.09,A -85,B 0,C 180,E1 -27539.739,E2 -27539.739} C_VEL
LIN {X 0,Y 193.334,Z 487.845,A -85,B 0,C 180,E1 -27540.354,E2 -27540.354} C_VEL
LIN {X 0,Y 190.441,Z 501.808,A -85,B 0,C 180,E1 -27540.783,E2 -27540.783} C_VEL
LIN {X 0,Y 186.369,Z 515.336,A -85,B 0,C 180,E1 -27541.409,E2 -27541.409} C_VEL
LIN {X 0,Y 181.888,Z 526.74,A -85,B 0,C 180,E1 -27542.071,E2 -27542.071} C_VEL
LIN {X 0,Y 175.939,Z 538.887,A -85,B 0,C 180,E1 -27543.037,E2 -27543.037} C_VEL
LIN {X 0,Y 169.125,Z 550.272,A -85,B 0,C 180,E1 -27544.231,E2 -27544.231} C_VEL
LIN {X 0,Y 160.7,Z 561.851,A -85,B 0,C 180,E1 -27545.794,E2 -27545.794} C_VEL
LIN {X 0,Y 152.447,Z 571.411,A -85,B 0,C 180,E1 -27547.53,E2 -27547.53} C_VEL
LIN {X 0,Y 142.68,Z 580.985,A -85,B 0,C 180,E1 -27549.906,E2 -27549.906} C_VEL
LIN {X 0,Y 132.647,Z 589.251,A -85,B 0,C 180,E1 -27552.777,E2 -27552.777} C_VEL
LIN {X 0,Y 124.103,Z 595.249,A -85,B 0,C 180,E1 -27555.708,E2 -27555.708} C_VEL
LIN {X 0,Y 115.409,Z 600.481,A -85,B 0,C 180,E1 -27559.295,E2 -27559.295} C_VEL
LIN {X 0,Y 107.241,Z 604.631,A -85,B 0,C 180,E1 -27563.449,E2 -27563.449} C_VEL
LIN {X 0,Y 102.161,Z 606.845,A -85,B 0,C 180,E1 -27566.589,E2 -27566.589} C_VEL
LIN {X 0,Y 93.003,Z 610.007,A -85,B 0,C 180,E1 -27573.781,E2 -27573.781} C_VEL
LIN {X 0,Y 85.589,Z 611.635,A -85,B 0,C 180,E1 -27582.359,E2 -27582.359} C_VEL
LIN {X 0,Y 80.227,Z 611.783,A -85,B 0,C 180,E1 -27592.184,E2 -27592.184} C_VEL
LIN {X 0,Y 77.118,Z 610.479,A -85,B 0,C 180,E1 -27602.898,E2 -27602.898} C_VEL
LIN {X 0,Y 76.48,Z 609.279,A -85,B 0,C 180,E1 -27608.439,E2 -27608.439} C_VEL
LIN {X 0,Y 76.787,Z 605.742,A -85,B 0,C 180,E1 -27619.457,E2 -27619.457} C_VEL
LIN {X 0,Y 78.325,Z 602.114,A -85,B 0,C 180,E1 -27627.433,E2 -27627.433} C_VEL
LIN {X 0,Y 80.794,Z 597.543,A -85,B 0,C 180,E1 -27634.995,E2 -27634.995} C_VEL
LIN {X 0,Y 85.026,Z 590.949,A -85,B 0,C 180,E1 -27643.143,E2 -27643.143} C_VEL
LIN {X 0,Y 89.611,Z 584.196,A -85,B 0,C 180,E1 -27649.307,E2 -27649.307} C_VEL
LIN {X 0,Y 95.26,Z 575.709,A -85,B 0,C 180,E1 -27655.105,E2 -27655.105} C_VEL
LIN {X 0,Y 101.49,Z 565.698,A -85,B 0,C 180,E1 -27660.139,E2 -27660.139} C_VEL
LIN {X 0,Y 107.863,Z 554.531,A -85,B 0,C 180,E1 -27664.196,E2 -27664.196} C_VEL
LIN {X 0,Y 113.404,Z 543.418,A -85,B 0,C 180,E1 -27667.178,E2 -27667.178} C_VEL
LIN {X 0,Y 118.67,Z 531.027,A -85,B 0,C 180,E1 -27669.657,E2 -27669.657} C_VEL
LIN {X 0,Y 123.143,Z 517.954,A -85,B 0,C 180,E1 -27671.606,E2 -27671.606} C_VEL
LIN {X 0,Y 126.783,Z 504.087,A -85,B 0,C 180,E1 -27673.104,E2 -27673.104} C_VEL
LIN {X 0,Y 129.487,Z 489.794,A -85,B 0,C 180,E1 -27674.122,E2 -27674.122} C_VEL
LIN {X 0,Y 131.54,Z 471.716,A -85,B 0,C 180,E1 -27674.88,E2 -27674.88} C_VEL
LIN {X 0,Y 134.299,Z 442.206,A -85,B 0,C 180,E1 -27675.994,E2 -27675.994} C_VEL
LIN {X 0,Y 130.36,Z 432.876,A -85,B 0,C 180,E1 -27679.69,E2 -27679.69} C_VEL
LIN {X 0,Y 126.341,Z 424.689,A -85,B 0,C 180,E1 -27684.057,E2 -27684.057} C_VEL
LIN {X 0,Y 122.665,Z 418.042,A -85,B 0,C 180,E1 -27688.961,E2 -27688.961} C_VEL
LIN {X 0,Y 120.334,Z 414.202,A -85,B 0,C 180,E1 -27692.741,E2 -27692.741} C_VEL
LIN {X 0,Y 118.266,Z 410.647,A -85,B 0,C 180,E1 -27697.136,E2 -27697.136} C_VEL
LIN {X 0,Y 116.206,Z 407.597,A -85,B 0,C 180,E1 -27704.055,E2 -27704.055} C_VEL
LIN {X 0,Y 115.905,Z 405.924,A -85,B 0,C 180,E1 -27707.031,E2 -27707.031} C_VEL
LIN {X 0,Y 116.202,Z 405.957,A -85,B 0,C 180,E1 -27716.401,E2 -27716.401} C_VEL
LIN {X 0,Y 117.302,Z 409.169,A -85,B 0,C 180,E1 -27721.668,E2 -27721.668} C_VEL
LIN {X 0,Y 118.591,Z 410.846,A -85,B 0,C 180,E1 -27725.019,E2 -27725.019} C_VEL
LIN {X 0,Y 120.76,Z 414.456,A -85,B 0,C 180,E1 -27729.382,E2 -27729.382} C_VEL
LIN {X 0,Y 123.341,Z 419.17,A -85,B 0,C 180,E1 -27733.501,E2 -27733.501} C_VEL
LIN {X 0,Y 126.661,Z 425.219,A -85,B 0,C 180,E1 -27737.777,E2 -27737.777} C_VEL
LIN {X 0,Y 130.257,Z 432.666,A -85,B 0,C 180,E1 -27741.671,E2 -27741.671} C_VEL
LIN {X 0,Y 132.706,Z 440.677,A -85,B 0,C 180,E1 -27744.271,E2 -27744.271} C_VEL
LIN {X 0,Y 134.099,Z 445.918,A -85,B 0,C 180,E1 -27745.698,E2 -27745.698} C_VEL
LIN {X 0,Y 129.578,Z 492.617,A -85,B 0,C 180,E1 -27747.513,E2 -27747.513} C_VEL
LIN {X 0,Y 127.065,Z 506.631,A -85,B 0,C 180,E1 -27748.379,E2 -27748.379} C_VEL
LIN {X 0,Y 123.462,Z 520.846,A -85,B 0,C 180,E1 -27749.757,E2 -27749.757} C_VEL
LIN {X 0,Y 118.606,Z 534.833,A -85,B 0,C 180,E1 -27751.588,E2 -27751.588} C_VEL
LIN {X 0,Y 113.411,Z 547.195,A -85,B 0,C 180,E1 -27753.9,E2 -27753.9} C_VEL
LIN {X 0,Y 109.5,Z 555.315,A -85,B 0,C 180,E1 -27755.869,E2 -27755.869} C_VEL
LIN {X 0,Y 104.015,Z 565.47,A -85,B 0,C 180,E1 -27759.006,E2 -27759.006} C_VEL
LIN {X 0,Y 97.189,Z 576.597,A -85,B 0,C 180,E1 -27763.682,E2 -27763.682} C_VEL
LIN {X 0,Y 91.219,Z 585.789,A -85,B 0,C 180,E1 -27769.084,E2 -27769.084} C_VEL
LIN {X 0,Y 86.053,Z 593.403,A -85,B 0,C 180,E1 -27775.127,E2 -27775.127} C_VEL
LIN {X 0,Y 82.062,Z 599.747,A -85,B 0,C 180,E1 -27781.894,E2 -27781.894} C_VEL
LIN {X 0,Y 79.098,Z 604.95,A -85,B 0,C 180,E1 -27789.177,E2 -27789.177} C_VEL
LIN {X 0,Y 77.439,Z 609.111,A -85,B 0,C 180,E1 -27796.881,E2 -27796.881} C_VEL
LIN {X 0,Y 76.852,Z 612.372,A -85,B 0,C 180,E1 -27804.748,E2 -27804.748} C_VEL
LIN {X 0,Y 77.049,Z 614.053,A -85,B 0,C 180,E1 -27809.995,E2 -27809.995} C_VEL
LIN {X 0,Y 76.89,Z 615.322,A -85,B 0,C 180,E1 -27815.24,E2 -27815.24} C_VEL
LIN {X 0,Y 77.946,Z 616.844,A -85,B 0,C 180,E1 -27825.689,E2 -27825.689} C_VEL
LIN {X 0,Y 81.199,Z 617.078,A -85,B 0,C 180,E1 -27835.638,E2 -27835.638} C_VEL
LIN {X 0,Y 86.731,Z 616.051,A -85,B 0,C 180,E1 -27844.552,E2 -27844.552} C_VEL
LIN {X 0,Y 94.071,Z 613.742,A -85,B 0,C 180,E1 -27852.246,E2 -27852.246} C_VEL
LIN {X 0,Y 102.928,Z 610.095,A -85,B 0,C 180,E1 -27858.679,E2 -27858.679} C_VEL
LIN {X 0,Y 112.917,Z 605.005,A -85,B 0,C 180,E1 -27864.004,E2 -27864.004} C_VEL
LIN {X 0,Y 123.877,Z 598.319,A -85,B 0,C 180,E1 -27868.315,E2 -27868.315} C_VEL
LIN {X 0,Y 133.935,Z 590.93,A -85,B 0,C 180,E1 -27871.507,E2 -27871.507} C_VEL
LIN {X 0,Y 144.362,Z 581.811,A -85,B 0,C 180,E1 -27874.235,E2 -27874.235} C_VEL
LIN {X 0,Y 153.573,Z 572.328,A -85,B 0,C 180,E1 -27876.236,E2 -27876.236} C_VEL
LIN {X 0,Y 162.215,Z 561.879,A -85,B 0,C 180,E1 -27877.824,E2 -27877.824} C_VEL
LIN {X 0,Y 169.375,Z 551.67,A -85,B 0,C 180,E1 -27878.997,E2 -27878.997} C_VEL
LIN {X 0,Y 176.65,Z 539.237,A -85,B 0,C 180,E1 -27880.03,E2 -27880.03} C_VEL
LIN {X 0,Y 182.316,Z 527.287,A -85,B 0,C 180,E1 -27880.803,E2 -27880.803} C_VEL
LIN {X 0,Y 187.066,Z 514.732,A -85,B 0,C 180,E1 -27881.369,E2 -27881.369} C_VEL
LIN {X 0,Y 188.135,Z 511.047,A -85,B 0,C 180,E1 -27881.703,E2 -27881.703} C_VEL
LIN {X 0,Y 190.323,Z 499.575,A -85,B 0,C 180,E1 -27883.755,E2 -27883.755} C_VEL
LIN {X 0,Y 190.999,Z 495.779,A -85,B 0,C 180,E1 -27884.063,E2 -27884.063} C_VEL
LIN {X 0,Y 191.324,Z 493.847,A -85,B 0,C 180,E1 -27884.19,E2 -27884.19} C_VEL
LIN {X 0,Y 191.025,Z 491.305,A -85,B 0,C 180,E1 -27886.299,E2 -27886.299} C_VEL
LIN {X 0,Y 190.537,Z 489.485,A -85,B 0,C 180,E1 -27890.98,E2 -27890.98} C_VEL
LIN {X 0,Y 190.554,Z 489.512,A -85,B 0,C 180,E1 -27892.285,E2 -27892.285} C_VEL
LIN {X 0,Y 190.966,Z 490.717,A -85,B 0,C 180,E1 -27895.988,E2 -27895.988} C_VEL
LIN {X 0,Y 191.386,Z 492.861,A -85,B 0,C 180,E1 -27898.369,E2 -27898.369} C_VEL
LIN {X 0,Y 187.965,Z 507.005,A -85,B 0,C 180,E1 -27898.854,E2 -27898.854} C_VEL
LIN {X 0,Y 183.254,Z 520.76,A -85,B 0,C 180,E1 -27899.491,E2 -27899.491} C_VEL
LIN {X 0,Y 177.685,Z 533.228,A -85,B 0,C 180,E1 -27900.287,E2 -27900.287} C_VEL
LIN {X 0,Y 171.341,Z 544.7,A -85,B 0,C 180,E1 -27901.252,E2 -27901.252} C_VEL
LIN {X 0,Y 163,Z 557.003,A -85,B 0,C 180,E1 -27902.624,E2 -27902.624} C_VEL
LIN {X 0,Y 154.995,Z 566.847,A -85,B 0,C 180,E1 -27904.049,E2 -27904.049} C_VEL
LIN {X 0,Y 144.888,Z 577.245,A -85,B 0,C 180,E1 -27906.106,E2 -27906.106} C_VEL
LIN {X 0,Y 135.002,Z 585.775,A -85,B 0,C 180,E1 -27908.485,E2 -27908.485} C_VEL
LIN {X 0,Y 125.391,Z 592.786,A -85,B 0,C 180,E1 -27911.247,E2 -27911.247} C_VEL
LIN {X 0,Y 116.106,Z 598.529,A -85,B 0,C 180,E1 -27914.436,E2 -27914.436} C_VEL
LIN {X 0,Y 107.264,Z 603.163,A -85,B 0,C 180,E1 -27918.199,E2 -27918.199} C_VEL
LIN {X 0,Y 98.954,Z 606.753,A -85,B 0,C 180,E1 -27922.598,E2 -27922.598} C_VEL
LIN {X 0,Y 91.938,Z 609.193,A -85,B 0,C 180,E1 -27927.299,E2 -27927.299} C_VEL
LIN {X 0,Y 84.551,Z 611.147,A -85,B 0,C 180,E1 -27933.785,E2 -27933.785} C_VEL
LIN {X 0,Y 80.63,Z 611.833,A -85,B 0,C 180,E1 -27938.336,E2 -27938.336} C_VEL
LIN {X 0,Y 74.351,Z 612.101,A -85,B 0,C 180,E1 -27948.579,E2 -27948.579} C_VEL
LIN {X 0,Y 70.486,Z 610.911,A -85,B 0,C 180,E1 -27960.103,E2 -27960.103} C_VEL
LIN {X 0,Y 69.581,Z 609.771,A -85,B 0,C 180,E1 -27966.176,E2 -27966.176} C_VEL
LIN {X 0,Y 69.496,Z 606.403,A -85,B 0,C 180,E1 -27978.336,E2 -27978.336} C_VEL
LIN {X 0,Y 71.127,Z 602.666,A -85,B 0,C 180,E1 -27987.537,E2 -27987.537} C_VEL
LIN {X 0,Y 73.607,Z 598.384,A -85,B 0,C 180,E1 -27995.484,E2 -27995.484} C_VEL
LIN {X 0,Y 78.013,Z 591.933,A -85,B 0,C 180,E1 -28004.349,E2 -28004.349} C_VEL
LIN {X 0,Y 83.35,Z 584.661,A -85,B 0,C 180,E1 -28011.515,E2 -28011.515} C_VEL
LIN {X 0,Y 89.888,Z 575.509,A -85,B 0,C 180,E1 -28017.981,E2 -28017.981} C_VEL
LIN {X 0,Y 96.542,Z 565.406,A -85,B 0,C 180,E1 -28023.096,E2 -28023.096} C_VEL
LIN {X 0,Y 103.287,Z 554.108,A -85,B 0,C 180,E1 -28027.153,E2 -28027.153} C_VEL
LIN {X 0,Y 109.1,Z 542.847,A -85,B 0,C 180,E1 -28030.108,E2 -28030.108} C_VEL
LIN {X 0,Y 114.475,Z 530.566,A -85,B 0,C 180,E1 -28032.483,E2 -28032.483} C_VEL
LIN {X 0,Y 118.739,Z 518.641,A -85,B 0,C 180,E1 -28034.226,E2 -28034.226} C_VEL
LIN {X 0,Y 122.616,Z 504.493,A -85,B 0,C 180,E1 -28035.738,E2 -28035.738} C_VEL
LIN {X 0,Y 125.467,Z 490.031,A -85,B 0,C 180,E1 -28036.739,E2 -28036.739} C_VEL
LIN {X 0,Y 127.684,Z 470.942,A -85,B 0,C 180,E1 -28037.521,E2 -28037.521} C_VEL
LIN {X 0,Y 130.188,Z 444.974,A -85,B 0,C 180,E1 -28038.498,E2 -28038.498} C_VEL
LIN {X 0,Y 126.718,Z 436.449,A -85,B 0,C 180,E1 -28042.216,E2 -28042.216} C_VEL
LIN {X 0,Y 123.597,Z 429.81,A -85,B 0,C 180,E1 -28046.075,E2 -28046.075} C_VEL
LIN {X 0,Y 120.641,Z 424.107,A -85,B 0,C 180,E1 -28050.463,E2 -28050.463} C_VEL
LIN {X 0,Y 118.705,Z 420.685,A -85,B 0,C 180,E1 -28053.943,E2 -28053.943} C_VEL
LIN {X 0,Y 117.022,Z 417.511,A -85,B 0,C 180,E1 -28057.883,E2 -28057.883} C_VEL
LIN {X 0,Y 115.108,Z 414.168,A -85,B 0,C 180,E1 -28065.337,E2 -28065.337} C_VEL
LIN {X 0,Y 114.958,Z 412.936,A -85,B 0,C 180,E1 -28067.533,E2 -28067.533} C_VEL
LIN {X 0,Y 115.191,Z 412.987,A -85,B 0,C 180,E1 -28075.764,E2 -28075.764} C_VEL
LIN {X 0,Y 116.375,Z 416.383,A -85,B 0,C 180,E1 -28081.681,E2 -28081.681} C_VEL
LIN {X 0,Y 117.275,Z 417.643,A -85,B 0,C 180,E1 -28084.153,E2 -28084.153} C_VEL
LIN {X 0,Y 119.581,Z 421.861,A -85,B 0,C 180,E1 -28089.104,E2 -28089.104} C_VEL
LIN {X 0,Y 122.487,Z 427.428,A -85,B 0,C 180,E1 -28093.816,E2 -28093.816} C_VEL
LIN {X 0,Y 125.474,Z 433.66,A -85,B 0,C 180,E1 -28097.779,E2 -28097.779} C_VEL
LIN {X 0,Y 127.577,Z 438.71,A -85,B 0,C 180,E1 -28100.245,E2 -28100.245} C_VEL
LIN {X 0,Y 130.038,Z 448.027,A -85,B 0,C 180,E1 -28103.181,E2 -28103.181} C_VEL
LIN {X 0,Y 125.55,Z 492.59,A -85,B 0,C 180,E1 -28104.901,E2 -28104.901} C_VEL
LIN {X 0,Y 122.897,Z 506.702,A -85,B 0,C 180,E1 -28105.747,E2 -28105.747} C_VEL
LIN {X 0,Y 119.339,Z 520.261,A -85,B 0,C 180,E1 -28107.029,E2 -28107.029} C_VEL
LIN {X 0,Y 114.308,Z 534.321,A -85,B 0,C 180,E1 -28108.815,E2 -28108.815} C_VEL
LIN {X 0,Y 108.782,Z 546.941,A -85,B 0,C 180,E1 -28111.123,E2 -28111.123} C_VEL
LIN {X 0,Y 104.153,Z 556.085,A -85,B 0,C 180,E1 -28113.375,E2 -28113.375} C_VEL
LIN {X 0,Y 99.015,Z 565.063,A -85,B 0,C 180,E1 -28116.153,E2 -28116.153} C_VEL
LIN {X 0,Y 92.364,Z 575.385,A -85,B 0,C 180,E1 -28120.451,E2 -28120.451} C_VEL
LIN {X 0,Y 85.916,Z 584.736,A -85,B 0,C 180,E1 -28125.943,E2 -28125.943} C_VEL
LIN {X 0,Y 80.296,Z 592.493,A -85,B 0,C 180,E1 -28132.211,E2 -28132.211} C_VEL
LIN {X 0,Y 75.816,Z 598.951,A -85,B 0,C 180,E1 -28139.342,E2 -28139.342} C_VEL
LIN {X 0,Y 72.452,Z 604.216,A -85,B 0,C 180,E1 -28147.164,E2 -28147.164} C_VEL
LIN {X 0,Y 70.507,Z 608.486,A -85,B 0,C 180,E1 -28155.565,E2 -28155.565} C_VEL
LIN {X 0,Y 69.775,Z 611.848,A -85,B 0,C 180,E1 -28164.214,E2 -28164.214} C_VEL
LIN {X 0,Y 69.953,Z 613.578,A -85,B 0,C 180,E1 -28169.995,E2 -28169.995} C_VEL
LIN {X 0,Y 69.829,Z 614.893,A -85,B 0,C 180,E1 -28175.771,E2 -28175.771} C_VEL
LIN {X 0,Y 71.104,Z 616.505,A -85,B 0,C 180,E1 -28187.243,E2 -28187.243} C_VEL
LIN {X 0,Y 74.836,Z 616.831,A -85,B 0,C 180,E1 -28198,E2 -28198} C_VEL
LIN {X 0,Y 80.951,Z 615.894,A -85,B 0,C 180,E1 -28207.419,E2 -28207.419} C_VEL
LIN {X 0,Y 88.922,Z 613.679,A -85,B 0,C 180,E1 -28215.336,E2 -28215.336} C_VEL
LIN {X 0,Y 98.376,Z 610.128,A -85,B 0,C 180,E1 -28221.792,E2 -28221.792} C_VEL
LIN {X 0,Y 108.885,Z 605.14,A -85,B 0,C 180,E1 -28227.037,E2 -28227.037} C_VEL
LIN {X 0,Y 120.301,Z 598.563,A -85,B 0,C 180,E1 -28231.192,E2 -28231.192} C_VEL
LIN {X 0,Y 130.7,Z 591.313,A -85,B 0,C 180,E1 -28234.24,E2 -28234.24} C_VEL
LIN {X 0,Y 141.432,Z 582.417,A -85,B 0,C 180,E1 -28236.816,E2 -28236.816} C_VEL
LIN {X 0,Y 150.874,Z 573.135,A -85,B 0,C 180,E1 -28238.683,E2 -28238.683} C_VEL
LIN {X 0,Y 159.696,Z 562.904,A -85,B 0,C 180,E1 -28240.159,E2 -28240.159} C_VEL
LIN {X 0,Y 167.809,Z 551.685,A -85,B 0,C 180,E1 -28241.354,E2 -28241.354} C_VEL
LIN {X 0,Y 175.204,Z 539.316,A -85,B 0,C 180,E1 -28242.297,E2 -28242.297} C_VEL
LIN {X 0,Y 181.791,Z 525.499,A -85,B 0,C 180,E1 -28243.095,E2 -28243.095} C_VEL
LIN {X 0,Y 186.978,Z 511.383,A -85,B 0,C 180,E1 -28243.626,E2 -28243.626} C_VEL
LIN {X 0,Y 190.737,Z 497.102,A -85,B 0,C 180,E1 -28244.033,E2 -28244.033} C_VEL
LIN {X 0,Y 190.999,Z 495.779,A -85,B 0,C 180,E1 -28244.063,E2 -28244.063} C_VEL
LIN {X 0,Y 191.151,Z 494.385,A -85,B 0,C 180,E1 -28244.346,E2 -28244.346} C_VEL
LIN {X 0,Y 191.043,Z 493.537,A -85,B 0,C 180,E1 -28245.017,E2 -28245.017} C_VEL
LIN {X 0,Y 190.619,Z 493.627,A -85,B 0,C 180,E1 -28246.148,E2 -28246.148} C_VEL
LIN {X 0,Y 189.261,Z 496.582,A -85,B 0,C 180,E1 -28249.45,E2 -28249.45} C_VEL
LIN {X 0,Y 189.136,Z 496.647,A -85,B 0,C 180,E1 -28250.457,E2 -28250.457} C_VEL
LIN {X 0,Y 189.158,Z 496.399,A -85,B 0,C 180,E1 -28251.99,E2 -28251.99} C_VEL
LIN {X 0,Y 189.416,Z 497.5,A -85,B 0,C 180,E1 -28255.567,E2 -28255.567} C_VEL
LIN {X 0,Y 189.464,Z 498.247,A -85,B 0,C 180,E1 -28256.404,E2 -28256.404} C_VEL
LIN {X 0,Y 185.391,Z 512.599,A -85,B 0,C 180,E1 -28256.914,E2 -28256.914} C_VEL
LIN {X 0,Y 180.255,Z 525.847,A -85,B 0,C 180,E1 -28257.547,E2 -28257.547} C_VEL
LIN {X 0,Y 174.007,Z 538.428,A -85,B 0,C 180,E1 -28258.348,E2 -28258.348} C_VEL
LIN {X 0,Y 166.921,Z 550.006,A -85,B 0,C 180,E1 -28259.372,E2 -28259.372} C_VEL
LIN {X 0,Y 158.133,Z 561.763,A -85,B 0,C 180,E1 -28260.681,E2 -28260.681} C_VEL
LIN {X 0,Y 149.444,Z 571.466,A -85,B 0,C 180,E1 -28262.168,E2 -28262.168} C_VEL
LIN {X 0,Y 139.163,Z 581.063,A -85,B 0,C 180,E1 -28264.168,E2 -28264.168} C_VEL
LIN {X 0,Y 129.481,Z 588.683,A -85,B 0,C 180,E1 -28266.402,E2 -28266.402} C_VEL
LIN {X 0,Y 120.865,Z 594.472,A -85,B 0,C 180,E1 -28268.719,E2 -28268.719} C_VEL
LIN {X 0,Y 111.295,Z 599.92,A -85,B 0,C 180,E1 -28271.842,E2 -28271.842} C_VEL
LIN {X 0,Y 100.674,Z 604.91,A -85,B 0,C 180,E1 -28276.213,E2 -28276.213} C_VEL
LIN {X 0,Y 90.703,Z 608.589,A -85,B 0,C 180,E1 -28281.607,E2 -28281.607} C_VEL
LIN {X 0,Y 80.537,Z 611.283,A -85,B 0,C 180,E1 -28289.243,E2 -28289.243} C_VEL
LIN {X 0,Y 72.156,Z 612.41,A -85,B 0,C 180,E1 -28298.821,E2 -28298.821} C_VEL
LIN {X 0,Y 66.082,Z 612.063,A -85,B 0,C 180,E1 -28310.356,E2 -28310.356} C_VEL
LIN {X 0,Y 62.738,Z 610.216,A -85,B 0,C 180,E1 -28323.653,E2 -28323.653} C_VEL
LIN {X 0,Y 62.242,Z 607.015,A -85,B 0,C 180,E1 -28336.954,E2 -28336.954} C_VEL
LIN {X 0,Y 63.448,Z 604.105,A -85,B 0,C 180,E1 -28345.471,E2 -28345.471} C_VEL
LIN {X 0,Y 66.419,Z 599.227,A -85,B 0,C 180,E1 -28356.079,E2 -28356.079} C_VEL
LIN {X 0,Y 71.057,Z 592.915,A -85,B 0,C 180,E1 -28365.788,E2 -28365.788} C_VEL
LIN {X 0,Y 77.236,Z 585.121,A -85,B 0,C 180,E1 -28374.082,E2 -28374.082} C_VEL
LIN {X 0,Y 83.598,Z 576.827,A -85,B 0,C 180,E1 -28380.297,E2 -28380.297} C_VEL
LIN {X 0,Y 90.625,Z 566.924,A -85,B 0,C 180,E1 -28385.57,E2 -28385.57} C_VEL
LIN {X 0,Y 97.671,Z 555.897,A -85,B 0,C 180,E1 -28389.693,E2 -28389.693} C_VEL
LIN {X 0,Y 104.42,Z 543.647,A -85,B 0,C 180,E1 -28392.962,E2 -28392.962} C_VEL
LIN {X 0,Y 110.268,Z 530.908,A -85,B 0,C 180,E1 -28395.383,E2 -28395.383} C_VEL
LIN {X 0,Y 114.974,Z 518.124,A -85,B 0,C 180,E1 -28397.187,E2 -28397.187} C_VEL
LIN {X 0,Y 118.859,Z 504.281,A -85,B 0,C 180,E1 -28398.612,E2 -28398.612} C_VEL
LIN {X 0,Y 121.729,Z 490.18,A -85,B 0,C 180,E1 -28399.535,E2 -28399.535} C_VEL
LIN {X 0,Y 124.117,Z 470.259,A -85,B 0,C 180,E1 -28400.308,E2 -28400.308} C_VEL
LIN {X 0,Y 126.346,Z 447.804,A -85,B 0,C 180,E1 -28401.15,E2 -28401.15} C_VEL
LIN {X 0,Y 123.359,Z 440.168,A -85,B 0,C 180,E1 -28404.844,E2 -28404.844} C_VEL
LIN {X 0,Y 120.455,Z 433.685,A -85,B 0,C 180,E1 -28409.063,E2 -28409.063} C_VEL
LIN {X 0,Y 118,Z 428.807,A -85,B 0,C 180,E1 -28413.348,E2 -28413.348} C_VEL
LIN {X 0,Y 117.039,Z 427.068,A -85,B 0,C 180,E1 -28415.364,E2 -28415.364} C_VEL
LIN {X 0,Y 115.655,Z 424.233,A -85,B 0,C 180,E1 -28419.038,E2 -28419.038} C_VEL
LIN {X 0,Y 114.039,Z 420.351,A -85,B 0,C 180,E1 -28427.328,E2 -28427.328} C_VEL
LIN {X 0,Y 114.027,Z 419.958,A -85,B 0,C 180,E1 -28427.97,E2 -28427.97} C_VEL
LIN {X 0,Y 114.216,Z 420.108,A -85,B 0,C 180,E1 -28435.321,E2 -28435.321} C_VEL
LIN {X 0,Y 115.322,Z 423.374,A -85,B 0,C 180,E1 -28441.272,E2 -28441.272} C_VEL
LIN {X 0,Y 115.94,Z 424.365,A -85,B 0,C 180,E1 -28443.14,E2 -28443.14} C_VEL
LIN {X 0,Y 117.987,Z 428.464,A -85,B 0,C 180,E1 -28448.01,E2 -28448.01} C_VEL
LIN {X 0,Y 120.45,Z 433.497,A -85,B 0,C 180,E1 -28452.365,E2 -28452.365} C_VEL
LIN {X 0,Y 122.951,Z 439.19,A -85,B 0,C 180,E1 -28456.075,E2 -28456.075} C_VEL
LIN {X 0,Y 124.701,Z 443.723,A -85,B 0,C 180,E1 -28458.378,E2 -28458.378} C_VEL
LIN {X 0,Y 126.246,Z 450.246,A -85,B 0,C 180,E1 -28460.521,E2 -28460.521} C_VEL
LIN {X 0,Y 121.732,Z 492.852,A -85,B 0,C 180,E1 -28462.12,E2 -28462.12} C_VEL
LIN {X 0,Y 119.006,Z 506.773,A -85,B 0,C 180,E1 -28462.935,E2 -28462.935} C_VEL
LIN {X 0,Y 115.134,Z 520.819,A -85,B 0,C 180,E1 -28464.236,E2 -28464.236} C_VEL
LIN {X 0,Y 110.299,Z 533.81,A -85,B 0,C 180,E1 -28465.833,E2 -28465.833} C_VEL
LIN {X 0,Y 104.542,Z 546.484,A -85,B 0,C 180,E1 -28468.074,E2 -28468.074} C_VEL
LIN {X 0,Y 99.603,Z 555.801,A -85,B 0,C 180,E1 -28470.309,E2 -28470.309} C_VEL
LIN {X 0,Y 94.287,Z 564.653,A -85,B 0,C 180,E1 -28473.006,E2 -28473.006} C_VEL
LIN {X 0,Y 87.88,Z 574.149,A -85,B 0,C 180,E1 -28476.89,E2 -28476.89} C_VEL
LIN {X 0,Y 80.903,Z 583.681,A -85,B 0,C 180,E1 -28482.4,E2 -28482.4} C_VEL
LIN {X 0,Y 74.781,Z 591.575,A -85,B 0,C 180,E1 -28488.857,E2 -28488.857} C_VEL
LIN {X 0,Y 69.711,Z 598.105,A -85,B 0,C 180,E1 -28496.318,E2 -28496.318} C_VEL
LIN {X 0,Y 65.911,Z 603.482,A -85,B 0,C 180,E1 -28504.748,E2 -28504.748} C_VEL
LIN {X 0,Y 63.171,Z 609.117,A -85,B 0,C 180,E1 -28517.138,E2 -28517.138} C_VEL
LIN {X 0,Y 62.705,Z 611.306,A -85,B 0,C 180,E1 -28523.559,E2 -28523.559} C_VEL
LIN {X 0,Y 62.849,Z 613.098,A -85,B 0,C 180,E1 -28529.994,E2 -28529.994} C_VEL
LIN {X 0,Y 62.756,Z 614.462,A -85,B 0,C 180,E1 -28536.424,E2 -28536.424} C_VEL
LIN {X 0,Y 64.333,Z 616.166,A -85,B 0,C 180,E1 -28549.125,E2 -28549.125} C_VEL
LIN {X 0,Y 68.625,Z 616.583,A -85,B 0,C 180,E1 -28560.794,E2 -28560.794} C_VEL
LIN {X 0,Y 75.389,Z 615.737,A -85,B 0,C 180,E1 -28570.728,E2 -28570.728} C_VEL
LIN {X 0,Y 84.059,Z 613.615,A -85,B 0,C 180,E1 -28578.798,E2 -28578.798} C_VEL
LIN {X 0,Y 94.137,Z 610.162,A -85,B 0,C 180,E1 -28585.201,E2 -28585.201} C_VEL
LIN {X 0,Y 105.185,Z 605.285,A -85,B 0,C 180,E1 -28590.289,E2 -28590.289} C_VEL
LIN {X 0,Y 117.05,Z 598.837,A -85,B 0,C 180,E1 -28594.235,E2 -28594.235} C_VEL
LIN {X 0,Y 127.782,Z 591.724,A -85,B 0,C 180,E1 -28597.1,E2 -28597.1} C_VEL
LIN {X 0,Y 137.215,Z 584.328,A -85,B 0,C 180,E1 -28599.178,E2 -28599.178} C_VEL
LIN {X 0,Y 146.853,Z 575.487,A -85,B 0,C 180,E1 -28600.933,E2 -28600.933} C_VEL
LIN {X 0,Y 154.986,Z 566.761,A -85,B 0,C 180,E1 -28602.216,E2 -28602.216} C_VEL
LIN {X 0,Y 164.033,Z 555.246,A -85,B 0,C 180,E1 -28603.458,E2 -28603.458} C_VEL
LIN {X 0,Y 171.535,Z 543.761,A -85,B 0,C 180,E1 -28604.318,E2 -28604.318} C_VEL
LIN {X 0,Y 178.2,Z 531.233,A -85,B 0,C 180,E1 -28605.063,E2 -28605.063} C_VEL
LIN {X 0,Y 184.084,Z 517.221,A -85,B 0,C 180,E1 -28605.62,E2 -28605.62} C_VEL
LIN {X 0,Y 188.563,Z 502.772,A -85,B 0,C 180,E1 -28606.028,E2 -28606.028} C_VEL
LIN {X 0,Y 189.52,Z 498.652,A -85,B 0,C 180,E1 -28606.174,E2 -28606.174} C_VEL
LIN {X 0,Y 189.443,Z 497.784,A -85,B 0,C 180,E1 -28607.138,E2 -28607.138} C_VEL
LIN {X 0,Y 189.136,Z 496.647,A -85,B 0,C 180,E1 -28610.457,E2 -28610.457} C_VEL
LIN {X 0,Y 188.998,Z 497.108,A -85,B 0,C 180,E1 -28611.466,E2 -28611.466} C_VEL
LIN {X 0,Y 188.55,Z 499.18,A -85,B 0,C 180,E1 -28612.548,E2 -28612.548} C_VEL
LIN {X 0,Y 187.986,Z 501.657,A -85,B 0,C 180,E1 -28613.29,E2 -28613.29} C_VEL
LIN {X 0,Y 186.674,Z 506.706,A -85,B 0,C 180,E1 -28614.224,E2 -28614.224} C_VEL
LIN {X 0,Y 185.435,Z 510.85,A -85,B 0,C 180,E1 -28614.637,E2 -28614.637} C_VEL
LIN {X 0,Y 184.959,Z 512.27,A -85,B 0,C 180,E1 -28614.704,E2 -28614.704} C_VEL
LIN {X 0,Y 179.647,Z 525.889,A -85,B 0,C 180,E1 -28615.284,E2 -28615.284} C_VEL
LIN {X 0,Y 173.481,Z 538.197,A -85,B 0,C 180,E1 -28615.991,E2 -28615.991} C_VEL
LIN {X 0,Y 166.271,Z 549.87,A -85,B 0,C 180,E1 -28616.91,E2 -28616.91} C_VEL
LIN {X 0,Y 158.222,Z 560.627,A -85,B 0,C 180,E1 -28617.964,E2 -28617.964} C_VEL
LIN {X 0,Y 149.35,Z 570.555,A -85,B 0,C 180,E1 -28619.26,E2 -28619.26} C_VEL
LIN {X 0,Y 138.819,Z 580.404,A -85,B 0,C 180,E1 -28621.047,E2 -28621.047} C_VEL
LIN {X 0,Y 128.361,Z 588.524,A -85,B 0,C 180,E1 -28623.138,E2 -28623.138} C_VEL
LIN {X 0,Y 116.594,Z 596.05,A -85,B 0,C 180,E1 -28626.004,E2 -28626.004} C_VEL
LIN {X 0,Y 106.727,Z 601.277,A -85,B 0,C 180,E1 -28629.001,E2 -28629.001} C_VEL
LIN {X 0,Y 97.501,Z 605.302,A -85,B 0,C 180,E1 -28632.487,E2 -28632.487} C_VEL
LIN {X 0,Y 88.16,Z 608.558,A -85,B 0,C 180,E1 -28636.953,E2 -28636.953} C_VEL
LIN {X 0,Y 77.082,Z 611.375,A -85,B 0,C 180,E1 -28644.263,E2 -28644.263} C_VEL
LIN {X 0,Y 67.624,Z 612.666,A -85,B 0,C 180,E1 -28653.765,E2 -28653.765} C_VEL
LIN {X 0,Y 60.423,Z 612.439,A -85,B 0,C 180,E1 -28665.752,E2 -28665.752} C_VEL
LIN {X 0,Y 56.131,Z 610.754,A -85,B 0,C 180,E1 -28679.953,E2 -28679.953} C_VEL
LIN {X 0,Y 55.055,Z 607.618,A -85,B 0,C 180,E1 -28695.215,E2 -28695.215} C_VEL
LIN {X 0,Y 56.352,Z 604.395,A -85,B 0,C 180,E1 -28706.093,E2 -28706.093} C_VEL
LIN {X 0,Y 59.209,Z 600.067,A -85,B 0,C 180,E1 -28716.823,E2 -28716.823} C_VEL
LIN {X 0,Y 63.337,Z 594.845,A -85,B 0,C 180,E1 -28726.111,E2 -28726.111} C_VEL
LIN {X 0,Y 68.792,Z 588.529,A -85,B 0,C 180,E1 -28734.126,E2 -28734.126} C_VEL
LIN {X 0,Y 75.214,Z 580.958,A -85,B 0,C 180,E1 -28740.931,E2 -28740.931} C_VEL
LIN {X 0,Y 82.39,Z 571.866,A -85,B 0,C 180,E1 -28746.668,E2 -28746.668} C_VEL
LIN {X 0,Y 90.224,Z 560.841,A -85,B 0,C 180,E1 -28751.466,E2 -28751.466} C_VEL
LIN {X 0,Y 97.176,Z 549.616,A -85,B 0,C 180,E1 -28754.846,E2 -28754.846} C_VEL
LIN {X 0,Y 103.661,Z 537.205,A -85,B 0,C 180,E1 -28757.507,E2 -28757.507} C_VEL
LIN {X 0,Y 109.255,Z 523.975,A -85,B 0,C 180,E1 -28759.578,E2 -28759.578} C_VEL
LIN {X 0,Y 113.959,Z 509.75,A -85,B 0,C 180,E1 -28761.137,E2 -28761.137} C_VEL
LIN {X 0,Y 117.417,Z 495.187,A -85,B 0,C 180,E1 -28762.256,E2 -28762.256} C_VEL
LIN {X 0,Y 119.503,Z 481.694,A -85,B 0,C 180,E1 -28762.888,E2 -28762.888} C_VEL
LIN {X 0,Y 122.807,Z 451.267,A -85,B 0,C 180,E1 -28763.862,E2 -28763.862} C_VEL
LIN {X 0,Y 121.758,Z 447.888,A -85,B 0,C 180,E1 -28765.377,E2 -28765.377} C_VEL
LIN {X 0,Y 119.168,Z 441.412,A -85,B 0,C 180,E1 -28769.356,E2 -28769.356} C_VEL
LIN {X 0,Y 116.75,Z 436.026,A -85,B 0,C 180,E1 -28773.824,E2 -28773.824} C_VEL
LIN {X 0,Y 115.639,Z 433.723,A -85,B 0,C 180,E1 -28776.367,E2 -28776.367} C_VEL
LIN {X 0,Y 114.394,Z 430.953,A -85,B 0,C 180,E1 -28780.063,E2 -28780.063} C_VEL
LIN {X 0,Y 113.093,Z 427.166,A -85,B 0,C 180,E1 -28788.217,E2 -28788.217} C_VEL
LIN {X 0,Y 113.209,Z 426.936,A -85,B 0,C 180,E1 -28794.251,E2 -28794.251} C_VEL
LIN {X 0,Y 114.662,Z 431.106,A -85,B 0,C 180,E1 -28802.158,E2 -28802.158} C_VEL
LIN {X 0,Y 116.463,Z 435.073,A -85,B 0,C 180,E1 -28806.933,E2 -28806.933} C_VEL
LIN {X 0,Y 118.457,Z 439.586,A -85,B 0,C 180,E1 -28810.855,E2 -28810.855} C_VEL
LIN {X 0,Y 120.638,Z 444.942,A -85,B 0,C 180,E1 -28814.444,E2 -28814.444} C_VEL
LIN {X 0,Y 121.956,Z 448.797,A -85,B 0,C 180,E1 -28816.425,E2 -28816.425} C_VEL
LIN {X 0,Y 122.779,Z 452.678,A -85,B 0,C 180,E1 -28817.769,E2 -28817.769} C_VEL
LIN {X 0,Y 118.391,Z 492.166,A -85,B 0,C 180,E1 -28819.132,E2 -28819.132} C_VEL
LIN {X 0,Y 115.56,Z 506.303,A -85,B 0,C 180,E1 -28819.905,E2 -28819.905} C_VEL
LIN {X 0,Y 111.606,Z 520.233,A -85,B 0,C 180,E1 -28821.122,E2 -28821.122} C_VEL
LIN {X 0,Y 106.607,Z 533.295,A -85,B 0,C 180,E1 -28822.632,E2 -28822.632} C_VEL
LIN {X 0,Y 100.632,Z 546.01,A -85,B 0,C 180,E1 -28824.775,E2 -28824.775} C_VEL
LIN {X 0,Y 95.96,Z 554.494,A -85,B 0,C 180,E1 -28826.673,E2 -28826.673} C_VEL
LIN {X 0,Y 89.197,Z 565.251,A -85,B 0,C 180,E1 -28829.914,E2 -28829.914} C_VEL
LIN {X 0,Y 82.459,Z 574.626,A -85,B 0,C 180,E1 -28833.792,E2 -28833.792} C_VEL
LIN {X 0,Y 75.066,Z 584.013,A -85,B 0,C 180,E1 -28839.423,E2 -28839.423} C_VEL
LIN {X 0,Y 68.231,Z 592.068,A -85,B 0,C 180,E1 -28846.426,E2 -28846.426} C_VEL
LIN {X 0,Y 62.286,Z 599.217,A -85,B 0,C 180,E1 -28855.648,E2 -28855.648} C_VEL
LIN {X 0,Y 58.412,Z 604.38,A -85,B 0,C 180,E1 -28865.088,E2 -28865.088} C_VEL
LIN {X 0,Y 56.239,Z 608.492,A -85,B 0,C 180,E1 -28875.52,E2 -28875.52} C_VEL
LIN {X 0,Y 55.633,Z 610.733,A -85,B 0,C 180,E1 -28882.736,E2 -28882.736} C_VEL
LIN {X 0,Y 55.753,Z 612.584,A -85,B 0,C 180,E1 -28889.993,E2 -28889.993} C_VEL
LIN {X 0,Y 55.713,Z 614.004,A -85,B 0,C 180,E1 -28897.24,E2 -28897.24} C_VEL
LIN {X 0,Y 57.637,Z 615.808,A -85,B 0,C 180,E1 -28911.45,E2 -28911.45} C_VEL
LIN {X 0,Y 62.587,Z 616.321,A -85,B 0,C 180,E1 -28924.149,E2 -28924.149} C_VEL
LIN {X 0,Y 70.124,Z 615.57,A -85,B 0,C 180,E1 -28934.545,E2 -28934.545} C_VEL
LIN {X 0,Y 79.531,Z 613.551,A -85,B 0,C 180,E1 -28942.677,E2 -28942.677} C_VEL
LIN {X 0,Y 90.252,Z 610.213,A -85,B 0,C 180,E1 -28948.926,E2 -28948.926} C_VEL
LIN {X 0,Y 101.85,Z 605.451,A -85,B 0,C 180,E1 -28953.763,E2 -28953.763} C_VEL
LIN {X 0,Y 114.141,Z 599.121,A -85,B 0,C 180,E1 -28957.448,E2 -28957.448} C_VEL
LIN {X 0,Y 125.2,Z 592.135,A -85,B 0,C 180,E1 -28960.084,E2 -28960.084} C_VEL
LIN {X 0,Y 136.488,Z 583.541,A -85,B 0,C 180,E1 -28962.277,E2 -28962.277} C_VEL
LIN {X 0,Y 146.347,Z 574.595,A -85,B 0,C 180,E1 -28963.823,E2 -28963.823} C_VEL
LIN {X 0,Y 156.317,Z 563.811,A -85,B 0,C 180,E1 -28965.147,E2 -28965.147} C_VEL
LIN {X 0,Y 164.705,Z 552.908,A -85,B 0,C 180,E1 -28966.096,E2 -28966.096} C_VEL
LIN {X 0,Y 172.301,Z 540.997,A -85,B 0,C 180,E1 -28966.855,E2 -28966.855} C_VEL
LIN {X 0,Y 179.074,Z 527.784,A -85,B 0,C 180,E1 -28967.476,E2 -28967.476} C_VEL
LIN {X 0,Y 184.505,Z 514.138,A -85,B 0,C 180,E1 -28967.907,E2 -28967.907} C_VEL
LIN {X 0,Y 187.532,Z 504.309,A -85,B 0,C 180,E1 -28968.198,E2 -28968.198} C_VEL
LIN {X 0,Y 187.448,Z 503.247,A -85,B 0,C 180,E1 -28971.374,E2 -28971.374} C_VEL
LIN {X 0,Y 187.508,Z 503.955,A -85,B 0,C 180,E1 -28974.421,E2 -28974.421} C_VEL
LIN {X 0,Y 184.959,Z 512.27,A -85,B 0,C 180,E1 -28974.704,E2 -28974.704} C_VEL
LIN {X 0,Y 182.953,Z 517.838,A -85,B 0,C 180,E1 -28974.718,E2 -28974.718} C_VEL
LIN {X 0,Y 179.095,Z 526.835,A -85,B 0,C 180,E1 -28974.214,E2 -28974.214} C_VEL
LIN {X 0,Y 174.654,Z 535.549,A -85,B 0,C 180,E1 -28973.719,E2 -28973.719} C_VEL
LIN {X 0,Y 171.712,Z 540.659,A -85,B 0,C 180,E1 -28973.771,E2 -28973.771} C_VEL
LIN {X 0,Y 164.115,Z 552.317,A -85,B 0,C 180,E1 -28974.624,E2 -28974.624} C_VEL
LIN {X 0,Y 155.051,Z 563.727,A -85,B 0,C 180,E1 -28975.672,E2 -28975.672} C_VEL
LIN {X 0,Y 145.298,Z 573.897,A -85,B 0,C 180,E1 -28976.973,E2 -28976.973} C_VEL
LIN {X 0,Y 135.329,Z 582.584,A -85,B 0,C 180,E1 -28978.488,E2 -28978.488} C_VEL
LIN {X 0,Y 124.743,Z 590.31,A -85,B 0,C 180,E1 -28980.409,E2 -28980.409} C_VEL
LIN {X 0,Y 112.605,Z 597.59,A -85,B 0,C 180,E1 -28983.092,E2 -28983.092} C_VEL
LIN {X 0,Y 102.443,Z 602.544,A -85,B 0,C 180,E1 -28985.911,E2 -28985.911} C_VEL
LIN {X 0,Y 92.591,Z 606.469,A -85,B 0,C 180,E1 -28989.366,E2 -28989.366} C_VEL
LIN {X 0,Y 86.233,Z 608.533,A -85,B 0,C 180,E1 -28992.062,E2 -28992.062} C_VEL
LIN {X 0,Y 74.252,Z 611.467,A -85,B 0,C 180,E1 -28998.841,E2 -28998.841} C_VEL
LIN {X 0,Y 63.68,Z 612.881,A -85,B 0,C 180,E1 -29008.017,E2 -29008.017} C_VEL
LIN {X 0,Y 55.242,Z 612.81,A -85,B 0,C 180,E1 -29020.252,E2 -29020.252} C_VEL
LIN {X 0,Y 49.726,Z 611.247,A -85,B 0,C 180,E1 -29035.583,E2 -29035.583} C_VEL
LIN {X 0,Y 48.343,Z 609.918,A -85,B 0,C 180,E1 -29044.151,E2 -29044.151} C_VEL
LIN {X 0,Y 48.456,Z 606.152,A -85,B 0,C 180,E1 -29061.668,E2 -29061.668} C_VEL
LIN {X 0,Y 50.859,Z 602.329,A -85,B 0,C 180,E1 -29073.969,E2 -29073.969} C_VEL
LIN {X 0,Y 54.808,Z 597.596,A -85,B 0,C 180,E1 -29084.867,E2 -29084.867} C_VEL
LIN {X 0,Y 61.251,Z 590.724,A -85,B 0,C 180,E1 -29095.492,E2 -29095.492} C_VEL
LIN {X 0,Y 67.977,Z 583.536,A -85,B 0,C 180,E1 -29102.879,E2 -29102.879} C_VEL
LIN {X 0,Y 75.478,Z 574.908,A -85,B 0,C 180,E1 -29108.946,E2 -29108.946} C_VEL
LIN {X 0,Y 83.577,Z 564.454,A -85,B 0,C 180,E1 -29113.933,E2 -29113.933} C_VEL
LIN {X 0,Y 91.512,Z 552.715,A -85,B 0,C 180,E1 -29117.667,E2 -29117.667} C_VEL
LIN {X 0,Y 98.195,Z 540.992,A -85,B 0,C 180,E1 -29120.305,E2 -29120.305} C_VEL
LIN {X 0,Y 104.084,Z 528.549,A -85,B 0,C 180,E1 -29122.307,E2 -29122.307} C_VEL
LIN {X 0,Y 109.237,Z 514.763,A -85,B 0,C 180,E1 -29123.929,E2 -29123.929} C_VEL
LIN {X 0,Y 113.165,Z 500.652,A -85,B 0,C 180,E1 -29125.092,E2 -29125.092} C_VEL
LIN {X 0,Y 115.78,Z 487.153,A -85,B 0,C 180,E1 -29125.771,E2 -29125.771} C_VEL
LIN {X 0,Y 119.552,Z 454.146,A -85,B 0,C 180,E1 -29126.825,E2 -29126.825} C_VEL
LIN {X 0,Y 117.533,Z 448.291,A -85,B 0,C 180,E1 -29130.262,E2 -29130.262} C_VEL
LIN {X 0,Y 115.218,Z 442.553,A -85,B 0,C 180,E1 -29134.981,E2 -29134.981} C_VEL
LIN {X 0,Y 114.157,Z 440.135,A -85,B 0,C 180,E1 -29137.726,E2 -29137.726} C_VEL
LIN {X 0,Y 113.231,Z 437.759,A -85,B 0,C 180,E1 -29140.889,E2 -29140.889} C_VEL
LIN {X 0,Y 112.173,Z 433.985,A -85,B 0,C 180,E1 -29149.168,E2 -29149.168} C_VEL
LIN {X 0,Y 112.283,Z 434.109,A -85,B 0,C 180,E1 -29154.102,E2 -29154.102} C_VEL
LIN {X 0,Y 113.459,Z 437.916,A -85,B 0,C 180,E1 -29161.293,E2 -29161.293} C_VEL
LIN {X 0,Y 115.044,Z 441.83,A -85,B 0,C 180,E1 -29165.981,E2 -29165.981} C_VEL
LIN {X 0,Y 117.524,Z 448.115,A -85,B 0,C 180,E1 -29171.144,E2 -29171.144} C_VEL
LIN {X 0,Y 119.219,Z 453.202,A -85,B 0,C 180,E1 -29174.118,E2 -29174.118} C_VEL
LIN {X 0,Y 119.555,Z 455.131,A -85,B 0,C 180,E1 -29174.802,E2 -29174.802} C_VEL
LIN {X 0,Y 115.2,Z 492.57,A -85,B 0,C 180,E1 -29176.028,E2 -29176.028} C_VEL
LIN {X 0,Y 112.225,Z 506.694,A -85,B 0,C 180,E1 -29176.749,E2 -29176.749} C_VEL
LIN {X 0,Y 108.042,Z 520.802,A -85,B 0,C 180,E1 -29177.939,E2 -29177.939} C_VEL
LIN {X 0,Y 102.487,Z 534.568,A -85,B 0,C 180,E1 -29179.446,E2 -29179.446} C_VEL
LIN {X 0,Y 96.534,Z 546.547,A -85,B 0,C 180,E1 -29181.397,E2 -29181.397} C_VEL
LIN {X 0,Y 91.023,Z 555.985,A -85,B 0,C 180,E1 -29183.516,E2 -29183.516} C_VEL
LIN {X 0,Y 85.108,Z 564.846,A -85,B 0,C 180,E1 -29186.091,E2 -29186.091} C_VEL
LIN {X 0,Y 77.31,Z 575.074,A -85,B 0,C 180,E1 -29190.267,E2 -29190.267} C_VEL
LIN {X 0,Y 69.465,Z 584.343,A -85,B 0,C 180,E1 -29195.956,E2 -29195.956} C_VEL
LIN {X 0,Y 62.614,Z 591.777,A -85,B 0,C 180,E1 -29202.628,E2 -29202.628} C_VEL
LIN {X 0,Y 56.496,Z 598.423,A -85,B 0,C 180,E1 -29211.531,E2 -29211.531} C_VEL
LIN {X 0,Y 52.007,Z 603.655,A -85,B 0,C 180,E1 -29221.765,E2 -29221.765} C_VEL
LIN {X 0,Y 49.338,Z 607.864,A -85,B 0,C 180,E1 -29233.44,E2 -29233.44} C_VEL
LIN {X 0,Y 48.587,Z 610.16,A -85,B 0,C 180,E1 -29241.676,E2 -29241.676} C_VEL
LIN {X 0,Y 48.647,Z 612.06,A -85,B 0,C 180,E1 -29249.993,E2 -29249.993} C_VEL
LIN {X 0,Y 48.659,Z 613.527,A -85,B 0,C 180,E1 -29258.297,E2 -29258.297} C_VEL
LIN {X 0,Y 51.046,Z 615.423,A -85,B 0,C 180,E1 -29274.388,E2 -29274.388} C_VEL
LIN {X 0,Y 56.814,Z 616.028,A -85,B 0,C 180,E1 -29288.199,E2 -29288.199} C_VEL
LIN {X 0,Y 65.22,Z 615.375,A -85,B 0,C 180,E1 -29298.956,E2 -29298.956} C_VEL
LIN {X 0,Y 75.418,Z 613.461,A -85,B 0,C 180,E1 -29306.992,E2 -29306.992} C_VEL
LIN {X 0,Y 86.787,Z 610.242,A -85,B 0,C 180,E1 -29312.961,E2 -29312.961} C_VEL
LIN {X 0,Y 98.916,Z 605.614,A -85,B 0,C 180,E1 -29317.455,E2 -29317.455} C_VEL
LIN {X 0,Y 111.61,Z 599.404,A -85,B 0,C 180,E1 -29320.817,E2 -29320.817} C_VEL
LIN {X 0,Y 122.971,Z 592.546,A -85,B 0,C 180,E1 -29323.182,E2 -29323.182} C_VEL
LIN {X 0,Y 134.509,Z 584.095,A -85,B 0,C 180,E1 -29325.14,E2 -29325.14} C_VEL
LIN {X 0,Y 144.539,Z 575.316,A -85,B 0,C 180,E1 -29326.512,E2 -29326.512} C_VEL
LIN {X 0,Y 154.666,Z 564.724,A -85,B 0,C 180,E1 -29327.664,E2 -29327.664} C_VEL
LIN {X 0,Y 163.157,Z 554.06,A -85,B 0,C 180,E1 -29328.495,E2 -29328.495} C_VEL
LIN {X 0,Y 170.839,Z 542.452,A -85,B 0,C 180,E1 -29329.151,E2 -29329.151} C_VEL
LIN {X 0,Y 177.687,Z 529.722,A -85,B 0,C 180,E1 -29329.683,E2 -29329.683} C_VEL
LIN {X 0,Y 183.386,Z 516.243,A -85,B 0,C 180,E1 -29330.06,E2 -29330.06} C_VEL
LIN {X 0,Y 184.793,Z 512.166,A -85,B 0,C 180,E1 -29330.146,E2 -29330.146} C_VEL
LIN {X 0,Y 185.363,Z 510.435,A -85,B 0,C 180,E1 -29330.313,E2 -29330.313} C_VEL
LIN {X 0,Y 185.383,Z 510.16,A -85,B 0,C 180,E1 -29331.931,E2 -29331.931} C_VEL
LIN {X 0,Y 185.379,Z 510.224,A -85,B 0,C 180,E1 -29332.375,E2 -29332.375} C_VEL
LIN {X 0,Y 180.797,Z 522.576,A -85,B 0,C 180,E1 -29332.865,E2 -29332.865} C_VEL
LIN {X 0,Y 175.081,Z 534.639,A -85,B 0,C 180,E1 -29333.441,E2 -29333.441} C_VEL
LIN {X 0,Y 171.712,Z 540.659,A -85,B 0,C 180,E1 -29333.771,E2 -29333.771} C_VEL
LIN {X 0,Y 168.584,Z 545.736,A -85,B 0,C 180,E1 -29333.853,E2 -29333.853} C_VEL
LIN {X 0,Y 162.884,Z 553.835,A -85,B 0,C 180,E1 -29333.448,E2 -29333.448} C_VEL
LIN {X 0,Y 156.797,Z 561.507,A -85,B 0,C 180,E1 -29333.064,E2 -29333.064} C_VEL
LIN {X 0,Y 152.925,Z 565.872,A -85,B 0,C 180,E1 -29333.209,E2 -29333.209} C_VEL
LIN {X 0,Y 143.008,Z 575.752,A -85,B 0,C 180,E1 -29334.358,E2 -29334.358} C_VEL
LIN {X 0,Y 132.119,Z 584.763,A -85,B 0,C 180,E1 -29335.819,E2 -29335.819} C_VEL
LIN {X 0,Y 122.605,Z 591.324,A -85,B 0,C 180,E1 -29337.321,E2 -29337.321} C_VEL
LIN {X 0,Y 112.451,Z 597.244,A -85,B 0,C 180,E1 -29339.216,E2 -29339.216} C_VEL
LIN {X 0,Y 101.94,Z 602.331,A -85,B 0,C 180,E1 -29341.628,E2 -29341.628} C_VEL
LIN {X 0,Y 91.654,Z 606.383,A -85,B 0,C 180,E1 -29344.617,E2 -29344.617} C_VEL
LIN {X 0,Y 78.448,Z 610.228,A -85,B 0,C 180,E1 -29349.811,E2 -29349.811} C_VEL
LIN {X 0,Y 66.12,Z 612.509,A -85,B 0,C 180,E1 -29356.959,E2 -29356.959} C_VEL
LIN {X 0,Y 55.246,Z 613.296,A -85,B 0,C 180,E1 -29367.08,E2 -29367.08} C_VEL
LIN {X 0,Y 46.715,Z 612.619,A -85,B 0,C 180,E1 -29381.229,E2 -29381.229} C_VEL
LIN {X 0,Y 41.739,Z 610.453,A -85,B 0,C 180,E1 -29399.669,E2 -29399.669} C_VEL
LIN {X 0,Y 41.15,Z 606.803,A -85,B 0,C 180,E1 -29420.175,E2 -29420.175} C_VEL
LIN {X 0,Y 43.586,Z 603.098,A -85,B 0,C 180,E1 -29434.633,E2 -29434.633} C_VEL
LIN {X 0,Y 47.859,Z 598.431,A -85,B 0,C 180,E1 -29447.087,E2 -29447.087} C_VEL
LIN {X 0,Y 54.833,Z 591.72,A -85,B 0,C 180,E1 -29458.735,E2 -29458.735} C_VEL
LIN {X 0,Y 63.365,Z 583.377,A -85,B 0,C 180,E1 -29467.598,E2 -29467.598} C_VEL
LIN {X 0,Y 71.454,Z 574.654,A -85,B 0,C 180,E1 -29473.518,E2 -29473.518} C_VEL
LIN {X 0,Y 80.056,Z 564.084,A -85,B 0,C 180,E1 -29478.269,E2 -29478.269} C_VEL
LIN {X 0,Y 88.382,Z 552.217,A -85,B 0,C 180,E1 -29481.749,E2 -29481.749} C_VEL
LIN {X 0,Y 95.355,Z 540.326,A -85,B 0,C 180,E1 -29484.174,E2 -29484.174} C_VEL
LIN {X 0,Y 101.648,Z 527.218,A -85,B 0,C 180,E1 -29486.072,E2 -29486.072} C_VEL
LIN {X 0,Y 106.786,Z 513.504,A -85,B 0,C 180,E1 -29487.49,E2 -29487.49} C_VEL
LIN {X 0,Y 110.584,Z 499.762,A -85,B 0,C 180,E1 -29488.484,E2 -29488.484} C_VEL
LIN {X 0,Y 113.249,Z 485.715,A -85,B 0,C 180,E1 -29489.09,E2 -29489.09} C_VEL
LIN {X 0,Y 116.535,Z 457.271,A -85,B 0,C 180,E1 -29489.978,E2 -29489.978} C_VEL
LIN {X 0,Y 114.691,Z 451.762,A -85,B 0,C 180,E1 -29493.791,E2 -29493.791} C_VEL
LIN {X 0,Y 113,Z 447.102,A -85,B 0,C 180,E1 -29498.306,E2 -29498.306} C_VEL
LIN {X 0,Y 111.983,Z 444.472,A -85,B 0,C 180,E1 -29502.145,E2 -29502.145} C_VEL
LIN {X 0,Y 111.261,Z 441.026,A -85,B 0,C 180,E1 -29509.771,E2 -29509.771} C_VEL
LIN {X 0,Y 111.343,Z 441.183,A -85,B 0,C 180,E1 -29513.661,E2 -29513.661} C_VEL
LIN {X 0,Y 112.256,Z 444.719,A -85,B 0,C 180,E1 -29520.328,E2 -29520.328} C_VEL
LIN {X 0,Y 113.515,Z 448.2,A -85,B 0,C 180,E1 -29524.609,E2 -29524.609} C_VEL
LIN {X 0,Y 115.547,Z 454.077,A -85,B 0,C 180,E1 -29529.493,E2 -29529.493} C_VEL
LIN {X 0,Y 116.633,Z 457.555,A -85,B 0,C 180,E1 -29531.651,E2 -29531.651} C_VEL
LIN {X 0,Y 112.552,Z 491.892,A -85,B 0,C 180,E1 -29532.716,E2 -29532.716} C_VEL
LIN {X 0,Y 109.627,Z 505.712,A -85,B 0,C 180,E1 -29533.349,E2 -29533.349} C_VEL
LIN {X 0,Y 105.234,Z 520.207,A -85,B 0,C 180,E1 -29534.435,E2 -29534.435} C_VEL
LIN {X 0,Y 99.517,Z 534.045,A -85,B 0,C 180,E1 -29535.79,E2 -29535.79} C_VEL
LIN {X 0,Y 93.128,Z 546.487,A -85,B 0,C 180,E1 -29537.635,E2 -29537.635} C_VEL
LIN {X 0,Y 87.618,Z 555.551,A -85,B 0,C 180,E1 -29539.515,E2 -29539.515} C_VEL
LIN {X 0,Y 81.439,Z 564.442,A -85,B 0,C 180,E1 -29541.909,E2 -29541.909} C_VEL
LIN {X 0,Y 72.503,Z 575.525,A -85,B 0,C 180,E1 -29546.269,E2 -29546.269} C_VEL
LIN {X 0,Y 64.153,Z 584.67,A -85,B 0,C 180,E1 -29551.884,E2 -29551.884} C_VEL
LIN {X 0,Y 57.326,Z 591.483,A -85,B 0,C 180,E1 -29558.105,E2 -29558.105} C_VEL
LIN {X 0,Y 51.05,Z 597.602,A -85,B 0,C 180,E1 -29566.492,E2 -29566.492} C_VEL
LIN {X 0,Y 45.812,Z 602.919,A -85,B 0,C 180,E1 -29577.516,E2 -29577.516} C_VEL
LIN {X 0,Y 42.538,Z 607.238,A -85,B 0,C 180,E1 -29590.696,E2 -29590.696} C_VEL
LIN {X 0,Y 41.554,Z 609.586,A -85,B 0,C 180,E1 -29600.254,E2 -29600.254} C_VEL
LIN {X 0,Y 41.541,Z 611.537,A -85,B 0,C 180,E1 -29609.991,E2 -29609.991} C_VEL
LIN {X 0,Y 41.629,Z 613.049,A -85,B 0,C 180,E1 -29619.711,E2 -29619.711} C_VEL
LIN {X 0,Y 44.637,Z 615.032,A -85,B 0,C 180,E1 -29638.177,E2 -29638.177} C_VEL
LIN {X 0,Y 51.39,Z 615.733,A -85,B 0,C 180,E1 -29653.13,E2 -29653.13} C_VEL
LIN {X 0,Y 60.753,Z 615.178,A -85,B 0,C 180,E1 -29664.062,E2 -29664.062} C_VEL
LIN {X 0,Y 71.78,Z 613.363,A -85,B 0,C 180,E1 -29671.775,E2 -29671.775} C_VEL
LIN {X 0,Y 83.791,Z 610.246,A -85,B 0,C 180,E1 -29677.302,E2 -29677.302} C_VEL
LIN {X 0,Y 96.418,Z 605.738,A -85,B 0,C 180,E1 -29681.353,E2 -29681.353} C_VEL
LIN {X 0,Y 109.482,Z 599.687,A -85,B 0,C 180,E1 -29684.33,E2 -29684.33} C_VEL
LIN {X 0,Y 121.115,Z 592.957,A -85,B 0,C 180,E1 -29686.386,E2 -29686.386} C_VEL
LIN {X 0,Y 132.87,Z 584.651,A -85,B 0,C 180,E1 -29688.092,E2 -29688.092} C_VEL
LIN {X 0,Y 143.058,Z 576.036,A -85,B 0,C 180,E1 -29689.261,E2 -29689.261} C_VEL
LIN {X 0,Y 153.315,Z 565.639,A -85,B 0,C 180,E1 -29690.237,E2 -29690.237} C_VEL
LIN {X 0,Y 161.899,Z 555.216,A -85,B 0,C 180,E1 -29690.941,E2 -29690.941} C_VEL
LIN {X 0,Y 166.284,Z 549.085,A -85,B 0,C 180,E1 -29691.238,E2 -29691.238} C_VEL
LIN {X 0,Y 167.126,Z 547.794,A -85,B 0,C 180,E1 -29691.811,E2 -29691.811} C_VEL
LIN {X 0,Y 158.231,Z 559.748,A -85,B 0,C 180,E1 -29692.672,E2 -29692.672} C_VEL
LIN {X 0,Y 152.925,Z 565.872,A -85,B 0,C 180,E1 -29693.209,E2 -29693.209} C_VEL
LIN {X 0,Y 148.837,Z 570.214,A -85,B 0,C 180,E1 -29693.377,E2 -29693.377} C_VEL
LIN {X 0,Y 141.563,Z 577.059,A -85,B 0,C 180,E1 -29693.03,E2 -29693.03} C_VEL
LIN {X 0,Y 133.86,Z 583.375,A -85,B 0,C 180,E1 -29692.719,E2 -29692.719} C_VEL
LIN {X 0,Y 129.096,Z 586.866,A -85,B 0,C 180,E1 -29693.014,E2 -29693.014} C_VEL
LIN {X 0,Y 116.44,Z 594.905,A -85,B 0,C 180,E1 -29694.766,E2 -29694.766} C_VEL
LIN {X 0,Y 105.596,Z 600.485,A -85,B 0,C 180,E1 -29696.628,E2 -29696.628} C_VEL
LIN {X 0,Y 94.887,Z 604.975,A -85,B 0,C 180,E1 -29698.948,E2 -29698.948} C_VEL
LIN {X 0,Y 84.373,Z 608.479,A -85,B 0,C 180,E1 -29701.846,E2 -29701.846} C_VEL
LIN {X 0,Y 70.805,Z 611.65,A -85,B 0,C 180,E1 -29707.028,E2 -29707.028} C_VEL
LIN {X 0,Y 58.073,Z 613.292,A -85,B 0,C 180,E1 -29714.524,E2 -29714.524} C_VEL
LIN {X 0,Y 46.829,Z 613.456,A -85,B 0,C 180,E1 -29725.798,E2 -29725.798} C_VEL
LIN {X 0,Y 38.185,Z 612.165,A -85,B 0,C 180,E1 -29742.605,E2 -29742.605} C_VEL
LIN {X 0,Y 35.462,Z 610.969,A -85,B 0,C 180,E1 -29753.532,E2 -29753.532} C_VEL
LIN {X 0,Y 33.914,Z 609.405,A -85,B 0,C 180,E1 -29765.527,E2 -29765.527} C_VEL
LIN {X 0,Y 34.422,Z 606.209,A -85,B 0,C 180,E1 -29784.739,E2 -29784.739} C_VEL
LIN {X 0,Y 37.647,Z 602.375,A -85,B 0,C 180,E1 -29800.769,E2 -29800.769} C_VEL
LIN {X 0,Y 42.977,Z 597.526,A -85,B 0,C 180,E1 -29814.14,E2 -29814.14} C_VEL
LIN {X 0,Y 51.155,Z 590.498,A -85,B 0,C 180,E1 -29825.73,E2 -29825.73} C_VEL
LIN {X 0,Y 60.613,Z 581.795,A -85,B 0,C 180,E1 -29834.09,E2 -29834.09} C_VEL
LIN {X 0,Y 69.39,Z 572.704,A -85,B 0,C 180,E1 -29839.438,E2 -29839.438} C_VEL
LIN {X 0,Y 78.6,Z 561.681,A -85,B 0,C 180,E1 -29843.591,E2 -29843.591} C_VEL
LIN {X 0,Y 86.524,Z 550.469,A -85,B 0,C 180,E1 -29846.37,E2 -29846.37} C_VEL
LIN {X 0,Y 93.954,Z 537.771,A -85,B 0,C 180,E1 -29848.505,E2 -29848.505} C_VEL
LIN {X 0,Y 99.477,Z 526.182,A -85,B 0,C 180,E1 -29849.941,E2 -29849.941} C_VEL
LIN {X 0,Y 104.359,Z 513.258,A -85,B 0,C 180,E1 -29851.108,E2 -29851.108} C_VEL
LIN {X 0,Y 108.216,Z 499.527,A -85,B 0,C 180,E1 -29851.988,E2 -29851.988} C_VEL
LIN {X 0,Y 110.901,Z 485.434,A -85,B 0,C 180,E1 -29852.53,E2 -29852.53} C_VEL
LIN {X 0,Y 113.854,Z 460.803,A -85,B 0,C 180,E1 -29853.198,E2 -29853.198} C_VEL
LIN {X 0,Y 112.186,Z 455.278,A -85,B 0,C 180,E1 -29857.737,E2 -29857.737} C_VEL
LIN {X 0,Y 111.162,Z 452.189,A -85,B 0,C 180,E1 -29861.573,E2 -29861.573} C_VEL
LIN {X 0,Y 110.657,Z 450.782,A -85,B 0,C 180,E1 -29864.261,E2 -29864.261} C_VEL
LIN {X 0,Y 110.359,Z 448.067,A -85,B 0,C 180,E1 -29870.384,E2 -29870.384} C_VEL
LIN {X 0,Y 110.406,Z 448.243,A -85,B 0,C 180,E1 -29873.147,E2 -29873.147} C_VEL
LIN {X 0,Y 111.101,Z 451.462,A -85,B 0,C 180,E1 -29879.368,E2 -29879.368} C_VEL
LIN {X 0,Y 112.206,Z 455.05,A -85,B 0,C 180,E1 -29883.699,E2 -29883.699} C_VEL
LIN {X 0,Y 113.911,Z 460.845,A -85,B 0,C 180,E1 -29888.356,E2 -29888.356} C_VEL
LIN {X 0,Y 112.934,Z 469.751,A -85,B 0,C 180,E1 -29888.685,E2 -29888.685} C_VEL
LIN {X 0,Y 109.89,Z 493.087,A -85,B 0,C 180,E1 -29889.331,E2 -29889.331} C_VEL
LIN {X 0,Y 106.793,Z 506.78,A -85,B 0,C 180,E1 -29889.89,E2 -29889.89} C_VEL
LIN {X 0,Y 102.424,Z 520.581,A -85,B 0,C 180,E1 -29890.848,E2 -29890.848} C_VEL
LIN {X 0,Y 96.978,Z 533.385,A -85,B 0,C 180,E1 -29891.928,E2 -29891.928} C_VEL
LIN {X 0,Y 90.324,Z 546.014,A -85,B 0,C 180,E1 -29893.565,E2 -29893.565} C_VEL
LIN {X 0,Y 84.673,Z 555.019,A -85,B 0,C 180,E1 -29895.212,E2 -29895.212} C_VEL
LIN {X 0,Y 77.451,Z 564.953,A -85,B 0,C 180,E1 -29897.662,E2 -29897.662} C_VEL
LIN {X 0,Y 69.619,Z 574.249,A -85,B 0,C 180,E1 -29900.955,E2 -29900.955} C_VEL
LIN {X 0,Y 60.668,Z 583.568,A -85,B 0,C 180,E1 -29906.118,E2 -29906.118} C_VEL
LIN {X 0,Y 52.468,Z 591.149,A -85,B 0,C 180,E1 -29912.706,E2 -29912.706} C_VEL
LIN {X 0,Y 43.89,Z 598.65,A -85,B 0,C 180,E1 -29923.887,E2 -29923.887} C_VEL
LIN {X 0,Y 38.323,Z 603.768,A -85,B 0,C 180,E1 -29936.61,E2 -29936.61} C_VEL
LIN {X 0,Y 35.074,Z 607.847,A -85,B 0,C 180,E1 -29952.498,E2 -29952.498} C_VEL
LIN {X 0,Y 34.428,Z 610.996,A -85,B 0,C 180,E1 -29969.989,E2 -29969.989} C_VEL
LIN {X 0,Y 34.65,Z 612.558,A -85,B 0,C 180,E1 -29981.692,E2 -29981.692} C_VEL
LIN {X 0,Y 38.495,Z 614.639,A -85,B 0,C 180,E1 -30003.198,E2 -30003.198} C_VEL
LIN {X 0,Y 46.438,Z 615.438,A -85,B 0,C 180,E1 -30019.162,E2 -30019.162} C_VEL
LIN {X 0,Y 56.846,Z 614.98,A -85,B 0,C 180,E1 -30029.917,E2 -30029.917} C_VEL
LIN {X 0,Y 68.692,Z 613.266,A -85,B 0,C 180,E1 -30037.029,E2 -30037.029} C_VEL
LIN {X 0,Y 81.31,Z 610.25,A -85,B 0,C 180,E1 -30041.934,E2 -30041.934} C_VEL
LIN {X 0,Y 94.39,Z 605.849,A -85,B 0,C 180,E1 -30045.435,E2 -30045.435} C_VEL
LIN {X 0,Y 107.78,Z 599.933,A -85,B 0,C 180,E1 -30047.97,E2 -30047.97} C_VEL
LIN {X 0,Y 120.378,Z 592.888,A -85,B 0,C 180,E1 -30049.774,E2 -30049.774} C_VEL
LIN {X 0,Y 131.594,Z 585.203,A -85,B 0,C 180,E1 -30051.104,E2 -30051.104} C_VEL
LIN {X 0,Y 135.028,Z 582.514,A -85,B 0,C 180,E1 -30051.442,E2 -30051.442} C_VEL
LIN {X 0,Y 137.394,Z 580.594,A -85,B 0,C 180,E1 -30052.036,E2 -30052.036} C_VEL
LIN {X 0,Y 129.096,Z 586.866,A -85,B 0,C 180,E1 -30053.014,E2 -30053.014} C_VEL
LIN {X 0,Y 123.506,Z 590.656,A -85,B 0,C 180,E1 -30053.434,E2 -30053.434} C_VEL
LIN {X 0,Y 113.706,Z 596.457,A -85,B 0,C 180,E1 -30053.351,E2 -30053.351} C_VEL
LIN {X 0,Y 105.595,Z 600.513,A -85,B 0,C 180,E1 -30053.254,E2 -30053.254} C_VEL
LIN {X 0,Y 99.435,Z 603.209,A -85,B 0,C 180,E1 -30053.662,E2 -30053.662} C_VEL
LIN {X 0,Y 97.405,Z 604.009,A -85,B 0,C 180,E1 -30053.972,E2 -30053.972} C_VEL
LIN {X 0,Y 84.474,Z 608.405,A -85,B 0,C 180,E1 -30056.643,E2 -30056.643} C_VEL
LIN {X 0,Y 72.606,Z 611.279,A -85,B 0,C 180,E1 -30059.998,E2 -30059.998} C_VEL
LIN {X 0,Y 63.368,Z 612.806,A -85,B 0,C 180,E1 -30063.568,E2 -30063.568} C_VEL
LIN {X 0,Y 50.156,Z 613.82,A -85,B 0,C 180,E1 -30071.267,E2 -30071.267} C_VEL
LIN {X 0,Y 38.415,Z 613.364,A -85,B 0,C 180,E1 -30083.855,E2 -30083.855} C_VEL
LIN {X 0,Y 29.522,Z 611.38,A -85,B 0,C 180,E1 -30105.569,E2 -30105.569} C_VEL
LIN {X 0,Y 26.629,Z 608.081,A -85,B 0,C 180,E1 -30134.711,E2 -30134.711} C_VEL
LIN {X 0,Y 29.238,Z 604.309,A -85,B 0,C 180,E1 -30157.935,E2 -30157.935} C_VEL
LIN {X 0,Y 34.284,Z 600.051,A -85,B 0,C 180,E1 -30174.215,E2 -30174.215} C_VEL
LIN {X 0,Y 42.747,Z 593.602,A -85,B 0,C 180,E1 -30188.073,E2 -30188.073} C_VEL
LIN {X 0,Y 50.506,Z 587.442,A -85,B 0,C 180,E1 -30195.546,E2 -30195.546} C_VEL
LIN {X 0,Y 60.282,Z 578.709,A -85,B 0,C 180,E1 -30201.911,E2 -30201.911} C_VEL
LIN {X 0,Y 69.718,Z 568.914,A -85,B 0,C 180,E1 -30206.277,E2 -30206.277} C_VEL
LIN {X 0,Y 78.664,Z 558.017,A -85,B 0,C 180,E1 -30209.315,E2 -30209.315} C_VEL
LIN {X 0,Y 86.935,Z 545.928,A -85,B 0,C 180,E1 -30211.549,E2 -30211.549} C_VEL
LIN {X 0,Y 94,Z 533.259,A -85,B 0,C 180,E1 -30213.187,E2 -30213.187} C_VEL
LIN {X 0,Y 99.865,Z 519.975,A -85,B 0,C 180,E1 -30214.387,E2 -30214.387} C_VEL
LIN {X 0,Y 104.603,Z 505.747,A -85,B 0,C 180,E1 -30215.3,E2 -30215.3} C_VEL
LIN {X 0,Y 107.795,Z 492.182,A -85,B 0,C 180,E1 -30215.898,E2 -30215.898} C_VEL
LIN {X 0,Y 110.511,Z 473,A -85,B 0,C 180,E1 -30216.368,E2 -30216.368} C_VEL
LIN {X 0,Y 111.48,Z 464.494,A -85,B 0,C 180,E1 -30216.661,E2 -30216.661} C_VEL
LIN {X 0,Y 110.427,Z 460.334,A -85,B 0,C 180,E1 -30220.597,E2 -30220.597} C_VEL
LIN {X 0,Y 109.746,Z 457.958,A -85,B 0,C 180,E1 -30224.242,E2 -30224.242} C_VEL
LIN {X 0,Y 109.45,Z 455.255,A -85,B 0,C 180,E1 -30230.304,E2 -30230.304} C_VEL
LIN {X 0,Y 109.48,Z 455.398,A -85,B 0,C 180,E1 -30232.857,E2 -30232.857} C_VEL
LIN {X 0,Y 109.972,Z 458.315,A -85,B 0,C 180,E1 -30238.424,E2 -30238.424} C_VEL
LIN {X 0,Y 110.746,Z 461.247,A -85,B 0,C 180,E1 -30242.091,E2 -30242.091} C_VEL
LIN {X 0,Y 111.574,Z 464.722,A -85,B 0,C 180,E1 -30245.051,E2 -30245.051} C_VEL
LIN {X 0,Y 108.037,Z 492.092,A -85,B 0,C 180,E1 -30245.718,E2 -30245.718} C_VEL
LIN {X 0,Y 104.939,Z 505.839,A -85,B 0,C 180,E1 -30246.189,E2 -30246.189} C_VEL
LIN {X 0,Y 100.461,Z 519.802,A -85,B 0,C 180,E1 -30246.986,E2 -30246.986} C_VEL
LIN {X 0,Y 94.901,Z 532.725,A -85,B 0,C 180,E1 -30247.88,E2 -30247.88} C_VEL
LIN {X 0,Y 87.904,Z 545.716,A -85,B 0,C 180,E1 -30249.282,E2 -30249.282} C_VEL
LIN {X 0,Y 82.239,Z 554.487,A -85,B 0,C 180,E1 -30250.629,E2 -30250.629} C_VEL
LIN {X 0,Y 74.753,Z 564.465,A -85,B 0,C 180,E1 -30252.711,E2 -30252.711} C_VEL
LIN {X 0,Y 65.774,Z 574.632,A -85,B 0,C 180,E1 -30255.9,E2 -30255.9} C_VEL
LIN {X 0,Y 56.315,Z 583.838,A -85,B 0,C 180,E1 -30260.595,E2 -30260.595} C_VEL
LIN {X 0,Y 47.331,Z 591.466,A -85,B 0,C 180,E1 -30266.997,E2 -30266.997} C_VEL
LIN {X 0,Y 39.255,Z 597.819,A -85,B 0,C 180,E1 -30276.311,E2 -30276.311} C_VEL
LIN {X 0,Y 32.576,Z 603.028,A -85,B 0,C 180,E1 -30289.653,E2 -30289.653} C_VEL
LIN {X 0,Y 28.358,Z 607.197,A -85,B 0,C 180,E1 -30308.163,E2 -30308.163} C_VEL
LIN {X 0,Y 27.338,Z 610.455,A -85,B 0,C 180,E1 -30329.987,E2 -30329.987} C_VEL
LIN {X 0,Y 27.743,Z 612.068,A -85,B 0,C 180,E1 -30344.661,E2 -30344.661} C_VEL
LIN {X 0,Y 32.764,Z 614.246,A -85,B 0,C 180,E1 -30370.039,E2 -30370.039} C_VEL
LIN {X 0,Y 42.121,Z 615.144,A -85,B 0,C 180,E1 -30386.524,E2 -30386.524} C_VEL
LIN {X 0,Y 55.168,Z 614.644,A -85,B 0,C 180,E1 -30397.529,E2 -30397.529} C_VEL
LIN {X 0,Y 66.239,Z 613.168,A -85,B 0,C 180,E1 -30402.708,E2 -30402.708} C_VEL
LIN {X 0,Y 79.388,Z 610.254,A -85,B 0,C 180,E1 -30406.834,E2 -30406.834} C_VEL
LIN {X 0,Y 92.856,Z 605.96,A -85,B 0,C 180,E1 -30409.692,E2 -30409.692} C_VEL
LIN {X 0,Y 106.525,Z 600.157,A -85,B 0,C 180,E1 -30411.711,E2 -30411.711} C_VEL
LIN {X 0,Y 106.866,Z 599.957,A -85,B 0,C 180,E1 -30412.441,E2 -30412.441} C_VEL
LIN {X 0,Y 97.405,Z 604.009,A -85,B 0,C 180,E1 -30413.972,E2 -30413.972} C_VEL
LIN {X 0,Y 91.943,Z 606.054,A -85,B 0,C 180,E1 -30414.585,E2 -30414.585} C_VEL
LIN {X 0,Y 82.47,Z 609.025,A -85,B 0,C 180,E1 -30414.567,E2 -30414.567} C_VEL
LIN {X 0,Y 72.833,Z 611.344,A -85,B 0,C 180,E1 -30414.567,E2 -30414.567} C_VEL
LIN {X 0,Y 67.132,Z 612.348,A -85,B 0,C 180,E1 -30415.49,E2 -30415.49} C_VEL
LIN {X 0,Y 54.295,Z 613.823,A -85,B 0,C 180,E1 -30419.997,E2 -30419.997} C_VEL
LIN {X 0,Y 42.464,Z 614.091,A -85,B 0,C 180,E1 -30426.851,E2 -30426.851} C_VEL
LIN {X 0,Y 30.055,Z 613.02,A -85,B 0,C 180,E1 -30440.75,E2 -30440.75} C_VEL
LIN {X 0,Y 23.777,Z 611.6,A -85,B 0,C 180,E1 -30456.233,E2 -30456.233} C_VEL
LIN {X 0,Y 19.537,Z 608.672,A -85,B 0,C 180,E1 -30488.937,E2 -30488.937} C_VEL
LIN {X 0,Y 21.207,Z 605.654,A -85,B 0,C 180,E1 -30516.225,E2 -30516.225} C_VEL
LIN {X 0,Y 27.833,Z 600.863,A -85,B 0,C 180,E1 -30540.347,E2 -30540.347} C_VEL
LIN {X 0,Y 37.343,Z 594.541,A -85,B 0,C 180,E1 -30554.903,E2 -30554.903} C_VEL
LIN {X 0,Y 46.621,Z 587.839,A -85,B 0,C 180,E1 -30562.556,E2 -30562.556} C_VEL
LIN {X 0,Y 56.129,Z 579.964,A -85,B 0,C 180,E1 -30567.703,E2 -30567.703} C_VEL
LIN {X 0,Y 66.013,Z 570.357,A -85,B 0,C 180,E1 -30571.452,E2 -30571.452} C_VEL
LIN {X 0,Y 75.243,Z 559.705,A -85,B 0,C 180,E1 -30574.039,E2 -30574.039} C_VEL
LIN {X 0,Y 83.757,Z 547.9,A -85,B 0,C 180,E1 -30575.864,E2 -30575.864} C_VEL
LIN {X 0,Y 91.438,Z 534.794,A -85,B 0,C 180,E1 -30577.278,E2 -30577.278} C_VEL
LIN {X 0,Y 97.853,Z 520.916,A -85,B 0,C 180,E1 -30578.319,E2 -30578.319} C_VEL
LIN {X 0,Y 102.682,Z 506.964,A -85,B 0,C 180,E1 -30579.06,E2 -30579.06} C_VEL
LIN {X 0,Y 106.08,Z 493.094,A -85,B 0,C 180,E1 -30579.591,E2 -30579.591} C_VEL
LIN {X 0,Y 108.376,Z 478.133,A -85,B 0,C 180,E1 -30579.9,E2 -30579.9} C_VEL
LIN {X 0,Y 109.524,Z 468.59,A -85,B 0,C 180,E1 -30580.131,E2 -30580.131} C_VEL
LIN {X 0,Y 108.997,Z 466.177,A -85,B 0,C 180,E1 -30582.937,E2 -30582.937} C_VEL
LIN {X 0,Y 108.655,Z 464.63,A -85,B 0,C 180,E1 -30585.557,E2 -30585.557} C_VEL
LIN {X 0,Y 108.527,Z 462.559,A -85,B 0,C 180,E1 -30590.22,E2 -30590.22} C_VEL
LIN {X 0,Y 108.553,Z 462.682,A -85,B 0,C 180,E1 -30592.796,E2 -30592.796} C_VEL
LIN {X 0,Y 108.87,Z 465.026,A -85,B 0,C 180,E1 -30597.354,E2 -30597.354} C_VEL
LIN {X 0,Y 109.426,Z 467.788,A -85,B 0,C 180,E1 -30600.737,E2 -30600.737} C_VEL
LIN {X 0,Y 109.582,Z 468.703,A -85,B 0,C 180,E1 -30601.54,E2 -30601.54} C_VEL
LIN {X 0,Y 106.372,Z 492.45,A -85,B 0,C 180,E1 -30602.033,E2 -30602.033} C_VEL
LIN {X 0,Y 103.138,Z 506.292,A -85,B 0,C 180,E1 -30602.409,E2 -30602.409} C_VEL
LIN {X 0,Y 98.538,Z 520.174,A -85,B 0,C 180,E1 -30603.058,E2 -30603.058} C_VEL
LIN {X 0,Y 93.318,Z 532.066,A -85,B 0,C 180,E1 -30603.673,E2 -30603.673} C_VEL
LIN {X 0,Y 86.376,Z 544.795,A -85,B 0,C 180,E1 -30604.734,E2 -30604.734} C_VEL
LIN {X 0,Y 81.216,Z 552.75,A -85,B 0,C 180,E1 -30605.602,E2 -30605.602} C_VEL
LIN {X 0,Y 72.653,Z 563.978,A -85,B 0,C 180,E1 -30607.433,E2 -30607.433} C_VEL
LIN {X 0,Y 64.177,Z 573.351,A -85,B 0,C 180,E1 -30609.71,E2 -30609.71} C_VEL
LIN {X 0,Y 54.209,Z 582.731,A -85,B 0,C 180,E1 -30613.479,E2 -30613.479} C_VEL
LIN {X 0,Y 44.536,Z 590.505,A -85,B 0,C 180,E1 -30618.744,E2 -30618.744} C_VEL
LIN {X 0,Y 35.48,Z 596.978,A -85,B 0,C 180,E1 -30626.933,E2 -30626.933} C_VEL
LIN {X 0,Y 27.51,Z 602.259,A -85,B 0,C 180,E1 -30639.948,E2 -30639.948} C_VEL
LIN {X 0,Y 21.883,Z 606.544,A -85,B 0,C 180,E1 -30661.182,E2 -30661.182} C_VEL
LIN {X 0,Y 20.23,Z 609.913,A -85,B 0,C 180,E1 -30689.982,E2 -30689.982} C_VEL
LIN {X 0,Y 20.943,Z 611.577,A -85,B 0,C 180,E1 -30709.589,E2 -30709.589} C_VEL
LIN {X 0,Y 27.68,Z 613.853,A -85,B 0,C 180,E1 -30739.595,E2 -30739.595} C_VEL
LIN {X 0,Y 38.648,Z 614.849,A -85,B 0,C 180,E1 -30755.375,E2 -30755.375} C_VEL
LIN {X 0,Y 51.919,Z 614.525,A -85,B 0,C 180,E1 -30764.29,E2 -30764.29} C_VEL
LIN {X 0,Y 64.479,Z 613.07,A -85,B 0,C 180,E1 -30768.772,E2 -30768.772} C_VEL
LIN {X 0,Y 78.074,Z 610.258,A -85,B 0,C 180,E1 -30771.931,E2 -30771.931} C_VEL
LIN {X 0,Y 77.897,Z 610.259,A -85,B 0,C 180,E1 -30772.91,E2 -30772.91} C_VEL
LIN {X 0,Y 67.132,Z 612.348,A -85,B 0,C 180,E1 -30775.49,E2 -30775.49} C_VEL
LIN {X 0,Y 61.416,Z 613.194,A -85,B 0,C 180,E1 -30776.598,E2 -30776.598} C_VEL
LIN {X 0,Y 51.559,Z 614.101,A -85,B 0,C 180,E1 -30777.051,E2 -30777.051} C_VEL
LIN {X 0,Y 41.664,Z 614.364,A -85,B 0,C 180,E1 -30777.692,E2 -30777.692} C_VEL
LIN {X 0,Y 35.948,Z 614.17,A -85,B 0,C 180,E1 -30779.885,E2 -30779.885} C_VEL
LIN {X 0,Y 28.269,Z 613.448,A -85,B 0,C 180,E1 -30786.163,E2 -30786.163} C_VEL
LIN {X 0,Y 16.343,Z 611.024,A -85,B 0,C 180,E1 -30810.72,E2 -30810.72} C_VEL
LIN {X 0,Y 12.433,Z 608.25,A -85,B 0,C 180,E1 -30853.612,E2 -30853.612} C_VEL
LIN {X 0,Y 16.609,Z 604.594,A -85,B 0,C 180,E1 -30895.057,E2 -30895.057} C_VEL
LIN {X 0,Y 24.813,Z 600.011,A -85,B 0,C 180,E1 -30915.101,E2 -30915.101} C_VEL
LIN {X 0,Y 35.895,Z 593.416,A -85,B 0,C 180,E1 -30926.335,E2 -30926.335} C_VEL
LIN {X 0,Y 47.589,Z 585.234,A -85,B 0,C 180,E1 -30932.401,E2 -30932.401} C_VEL
LIN {X 0,Y 57.786,Z 576.677,A -85,B 0,C 180,E1 -30935.819,E2 -30935.819} C_VEL
LIN {X 0,Y 68.084,Z 566.343,A -85,B 0,C 180,E1 -30938.297,E2 -30938.297} C_VEL
LIN {X 0,Y 76.754,Z 555.906,A -85,B 0,C 180,E1 -30939.821,E2 -30939.821} C_VEL
LIN {X 0,Y 84.572,Z 544.571,A -85,B 0,C 180,E1 -30940.974,E2 -30940.974} C_VEL
LIN {X 0,Y 91.846,Z 531.575,A -85,B 0,C 180,E1 -30941.879,E2 -30941.879} C_VEL
LIN {X 0,Y 97.267,Z 519.398,A -85,B 0,C 180,E1 -30942.521,E2 -30942.521} C_VEL
LIN {X 0,Y 102.177,Z 504.799,A -85,B 0,C 180,E1 -30943.094,E2 -30943.094} C_VEL
LIN {X 0,Y 105.523,Z 490.4,A -85,B 0,C 180,E1 -30943.418,E2 -30943.418} C_VEL
LIN {X 0,Y 107.845,Z 473.828,A -85,B 0,C 180,E1 -30943.678,E2 -30943.678} C_VEL
LIN {X 0,Y 107.904,Z 472.971,A -85,B 0,C 180,E1 -30943.908,E2 -30943.908} C_VEL
LIN {X 0,Y 107.651,Z 471.378,A -85,B 0,C 180,E1 -30946.581,E2 -30946.581} C_VEL
LIN {X 0,Y 107.608,Z 469.818,A -85,B 0,C 180,E1 -30950.136,E2 -30950.136} C_VEL
LIN {X 0,Y 107.632,Z 470.034,A -85,B 0,C 180,E1 -30952.97,E2 -30952.97} C_VEL
LIN {X 0,Y 107.83,Z 471.976,A -85,B 0,C 180,E1 -30956.569,E2 -30956.569} C_VEL
LIN {X 0,Y 107.99,Z 472.927,A -85,B 0,C 180,E1 -30957.937,E2 -30957.937} C_VEL
LIN {X 0,Y 105.045,Z 493.406,A -85,B 0,C 180,E1 -30958.264,E2 -30958.264} C_VEL
LIN {X 0,Y 101.803,Z 506.746,A -85,B 0,C 180,E1 -30958.518,E2 -30958.518} C_VEL
LIN {X 0,Y 97.095,Z 520.545,A -85,B 0,C 180,E1 -30958.993,E2 -30958.993} C_VEL
LIN {X 0,Y 91.374,Z 533.2,A -85,B 0,C 180,E1 -30959.438,E2 -30959.438} C_VEL
LIN {X 0,Y 84.342,Z 545.617,A -85,B 0,C 180,E1 -30960.131,E2 -30960.131} C_VEL
LIN {X 0,Y 76.449,Z 556.99,A -85,B 0,C 180,E1 -30961.086,E2 -30961.086} C_VEL
LIN {X 0,Y 66.846,Z 568.41,A -85,B 0,C 180,E1 -30962.7,E2 -30962.7} C_VEL
LIN {X 0,Y 56.435,Z 578.579,A -85,B 0,C 180,E1 -30964.884,E2 -30964.884} C_VEL
LIN {X 0,Y 46.165,Z 587.03,A -85,B 0,C 180,E1 -30968.275,E2 -30968.275} C_VEL
LIN {X 0,Y 34.475,Z 595.058,A -85,B 0,C 180,E1 -30974.421,E2 -30974.421} C_VEL
LIN {X 0,Y 23.562,Z 601.491,A -85,B 0,C 180,E1 -30986.482,E2 -30986.482} C_VEL
LIN {X 0,Y 16.006,Z 605.893,A -85,B 0,C 180,E1 -31008.774,E2 -31008.774} C_VEL
LIN {X 0,Y 13.141,Z 609.341,A -85,B 0,C 180,E1 -31049.972,E2 -31049.972} C_VEL
LIN {X 0,Y 14.436,Z 611.068,A -85,B 0,C 180,E1 -31079.104,E2 -31079.104} C_VEL
LIN {X 0,Y 23.687,Z 613.452,A -85,B 0,C 180,E1 -31112.852,E2 -31112.852} C_VEL
LIN {X 0,Y 36.258,Z 614.549,A -85,B 0,C 180,E1 -31125.694,E2 -31125.694} C_VEL
LIN {X 0,Y 49.689,Z 614.385,A -85,B 0,C 180,E1 -31131.866,E2 -31131.866} C_VEL
LIN {X 0,Y 49.5,Z 614.339,A -85,B 0,C 180,E1 -31133.574,E2 -31133.574} C_VEL
LIN {X 0,Y 35.948,Z 614.17,A -85,B 0,C 180,E1 -31139.885,E2 -31139.885} C_VEL
LIN {X 0,Y 30.296,Z 613.801,A -85,B 0,C 180,E1 -31142.809,E2 -31142.809} C_VEL
LIN {X 0,Y 20.549,Z 612.586,A -85,B 0,C 180,E1 -31146.079,E2 -31146.079} C_VEL
LIN {X 0,Y 12.814,Z 611.148,A -85,B 0,C 180,E1 -31151.104,E2 -31151.104} C_VEL
LIN {X 0,Y 7.64,Z 609.806,A -85,B 0,C 180,E1 -31166.341,E2 -31166.341} C_VEL
LIN {X 0,Y 6.369,Z 609.299,A -85,B 0,C 180,E1 -31178.227,E2 -31178.227} C_VEL
LIN {X 0,Y 10.418,Z 605.292,A -85,B 0,C 180,E1 -31272.472,E2 -31272.472} C_VEL
LIN {X 0,Y 20.36,Z 600.821,A -85,B 0,C 180,E1 -31289.684,E2 -31289.684} C_VEL
LIN {X 0,Y 32.459,Z 594.357,A -85,B 0,C 180,E1 -31296.986,E2 -31296.986} C_VEL
LIN {X 0,Y 44.713,Z 586.32,A -85,B 0,C 180,E1 -31300.599,E2 -31300.599} C_VEL
LIN {X 0,Y 55.233,Z 577.93,A -85,B 0,C 180,E1 -31302.634,E2 -31302.634} C_VEL
LIN {X 0,Y 65.771,Z 567.821,A -85,B 0,C 180,E1 -31304.111,E2 -31304.111} C_VEL
LIN {X 0,Y 75.467,Z 556.529,A -85,B 0,C 180,E1 -31305.075,E2 -31305.075} C_VEL
LIN {X 0,Y 83.397,Z 545.276,A -85,B 0,C 180,E1 -31305.74,E2 -31305.74} C_VEL
LIN {X 0,Y 90.208,Z 533.493,A -85,B 0,C 180,E1 -31306.25,E2 -31306.25} C_VEL
LIN {X 0,Y 96.28,Z 520.267,A -85,B 0,C 180,E1 -31306.672,E2 -31306.672} C_VEL
LIN {X 0,Y 101.253,Z 505.861,A -85,B 0,C 180,E1 -31307.04,E2 -31307.04} C_VEL
LIN {X 0,Y 104.801,Z 490.963,A -85,B 0,C 180,E1 -31307.283,E2 -31307.283} C_VEL
LIN {X 0,Y 106.683,Z 478.195,A -85,B 0,C 180,E1 -31307.512,E2 -31307.512} C_VEL
LIN {X 0,Y 106.705,Z 476.863,A -85,B 0,C 180,E1 -31311.119,E2 -31311.119} C_VEL
LIN {X 0,Y 106.719,Z 477.469,A -85,B 0,C 180,E1 -31313.385,E2 -31313.385} C_VEL
LIN {X 0,Y 106.746,Z 477.819,A -85,B 0,C 180,E1 -31314.179,E2 -31314.179} C_VEL
LIN {X 0,Y 104.16,Z 494.475,A -85,B 0,C 180,E1 -31314.405,E2 -31314.405} C_VEL
LIN {X 0,Y 100.916,Z 507.305,A -85,B 0,C 180,E1 -31314.536,E2 -31314.536} C_VEL
LIN {X 0,Y 96.155,Z 520.911,A -85,B 0,C 180,E1 -31314.82,E2 -31314.82} C_VEL
LIN {X 0,Y 89.773,Z 534.652,A -85,B 0,C 180,E1 -31315.044,E2 -31315.044} C_VEL
LIN {X 0,Y 83.136,Z 546.013,A -85,B 0,C 180,E1 -31315.334,E2 -31315.334} C_VEL
LIN {X 0,Y 74.88,Z 557.602,A -85,B 0,C 180,E1 -31315.795,E2 -31315.795} C_VEL
LIN {X 0,Y 65.123,Z 568.849,A -85,B 0,C 180,E1 -31316.698,E2 -31316.698} C_VEL
LIN {X 0,Y 54.512,Z 578.906,A -85,B 0,C 180,E1 -31317.826,E2 -31317.826} C_VEL
LIN {X 0,Y 43.754,Z 587.375,A -85,B 0,C 180,E1 -31319.699,E2 -31319.699} C_VEL
LIN {X 0,Y 31.677,Z 595.189,A -85,B 0,C 180,E1 -31323.047,E2 -31323.047} C_VEL
LIN {X 0,Y 21.353,Z 600.722,A -85,B 0,C 180,E1 -31329.002,E2 -31329.002} C_VEL
LIN {X 0,Y 11.627,Z 605.241,A -85,B 0,C 180,E1 -31344.876,E2 -31344.876} C_VEL
LIN {X 0,Y 6.027,Z 608.746,A -85,B 0,C 180,E1 -31409.94,E2 -31409.94} C_VEL
LIN {X 0,Y 8.924,Z 610.527,A -85,B 0,C 180,E1 -31461.887,E2 -31461.887} C_VEL
LIN {X 0,Y 21.393,Z 613.014,A -85,B 0,C 180,E1 -31490.147,E2 -31490.147} C_VEL
LIN {X 0,Y 21.157,Z 612.901,A -85,B 0,C 180,E1 -31495.021,E2 -31495.021} C_VEL
LIN {X 0,Y 14.074,Z 611.559,A -85,B 0,C 180,E1 -31503.368,E2 -31503.368} C_VEL
LIN {X 0,Y 6.369,Z 609.299,A -85,B 0,C 180,E1 -31538.227,E2 -31538.227} C_VEL
LIN {X 0,Y 6.519,Z 606.868,A -85,B 0,C 180,E1 -31617.563,E2 -31617.563} C_VEL
LIN {X 0,Y 12.786,Z 603.962,A -85,B 0,C 180,E1 -31650.415,E2 -31650.415} C_VEL
LIN {X 0,Y 22.584,Z 599.411,A -85,B 0,C 180,E1 -31664.367,E2 -31664.367} C_VEL
LIN {X 0,Y 32.597,Z 594,A -85,B 0,C 180,E1 -31669.106,E2 -31669.106} C_VEL
LIN {X 0,Y 37.525,Z 590.976,A -85,B 0,C 180,E1 -31669.575,E2 -31669.575} C_VEL
LIN {X 0,Y 48.2,Z 583.474,A -85,B 0,C 180,E1 -31669.845,E2 -31669.845} C_VEL
LIN {X 0,Y 58.862,Z 574.444,A -85,B 0,C 180,E1 -31670.107,E2 -31670.107} C_VEL
LIN {X 0,Y 64.151,Z 569.285,A -85,B 0,C 180,E1 -31670.426,E2 -31670.426} C_VEL
LIN {X 0,Y 53.47,Z 579.231,A -85,B 0,C 180,E1 -31670.367,E2 -31670.367} C_VEL
LIN {X 0,Y 41.969,Z 588.039,A -85,B 0,C 180,E1 -31670.363,E2 -31670.363} C_VEL
LIN {X 0,Y 30.325,Z 595.323,A -85,B 0,C 180,E1 -31670.116,E2 -31670.116} C_VEL
LIN {X 0,Y 28.541,Z 596.339,A -85,B 0,C 180,E1 -31670.119,E2 -31670.119} C_VEL
LIN {X 0,Y 28.582,Z 596.312,A -85,B 0,C 180,E1 -31669.661,E2 -31669.661} C_VEL
LIN {X 0,Y 37.525,Z 590.976,A -85,B 0,C 180,E1 -31669.575,E2 -31669.575} C_VEL
LIN {X 0,Y 40.603,Z 592.661,A -85,B 0,C 180,E1 -31669.538,E2 -31669.538} C_VEL
LIN {X 0,Y 40.603,Z 600,A -85,B 0,C 180,E1 -31669.538,E2 -31669.538} C_VEL
LIN {X 0,Y 40.603,Z 600,A -85,B 0,C 180,E1 -31669.538,E2 -31669.538}

QRS_NEXT_CUT()

QRS_NEXT()
QRS_HOME()

END
